       ELSE // illegal OPM              
           #FML_REF.OutData.FHPP[4] := 0;
           #Converted_BYTE5_8 := 0;
   END_CASE;

   (* Set Output DATA OF DRIVE *)
   #FML_REF.OutData.FHPP[5] := #BByte[1];
   #FML_REF.OutData.FHPP[6] := #BByte[2];
   #FML_REF.OutData.FHPP[7] := #BByte[3];
   #FML_REF.OutData.FHPP[8] := #BByte[4];
END_FUNCTION_BLOCK

FUNCTION_BLOCK "FB205_FHPP_SETIO_PART"   // FB205, SCL
TITLE = FHPPP SETIO_PART
{ S7_Optimized_Access := 'FALSE' }
AUTHOR : FESTO
FAMILY : E-DRIVE
VERSION : 5.1
// Set data from FHPP device using system function SETIO_PART
   VAR_INPUT
      ID : Word;
      Offset : Int;   // offset from start address where FHPP data start
   END_VAR
   VAR_OUTPUT
      Error : Bool;   // error while reading
      Status : "DT_FML_STATUS";
   END_VAR
   VAR_IN_OUT
      FML_REF : "DT_FML_REF";
   END_VAR
   VAR
      SET_PART : SETIO_PART;
   END_VAR
   VAR_TEMP
      i : Int;
      iByteCount : DInt;
      tmpFHPPplusSize : DInt;
      tmpFHPPplusElementSize : Array[1..9] of DInt;
      FHPPplus24 : Array[1..24] of Byte;
      WORD_BYTE : Word;
      WBYTE AT WORD_BYTE : Array[1..2] of Byte;
      DWORD_BYTE : DInt;
      DBYTE AT DWORD_BYTE : Array[1..4] of Byte;
      tmpStatus : "DT_FML_STATUS";
      tmp_FML_REF : "DT_FML_REF";
   END_VAR
BEGIN
   (*############################################################
       FESTO AG  Co., Esslingen
       Copyright (c) 2015. All rights reserved.    

       NAME OF FUNCTION BLOCK:         FHPP_SETIO_PART
       VERSION NUMBER:                 V5.1
       COMPOSER:                       bejk

   ############################################################*)

   // function block (FB) is busy
   #tmpStatus.Err := FALSE;
   #tmpStatus.Cat := 1;
   #tmpStatus.ID := 16#0000_0002; // FB busy 

   // ### FHPP Standard ###########################################
   #SET_PART(ID := #ID,
             OFFSET := #Offset,
             LEN := 8,
             ERROR => #tmpStatus.Err,
             OUTPUTS := #FML_REF.OutData.FHPP);

   // Error while writing
   IF #tmpStatus.Err THEN
       #tmpStatus.Cat := 4; // SIEMENS
       #tmpStatus.ID := DWORD_TO_DINT(#SET_PART.STATUS);
   END_IF;



   // ### EXIT ROUTINE ############################################################
   IF NOT #tmpStatus.Err THEN
       ENO := TRUE;      // Set ENO-Bit to true
       #Status := #tmpStatus;
       #Error := #tmpStatus.Err;
   ELSE
       ENO := FALSE;     // Set ENO-Bit to false
       #Status := #tmpStatus;
       #Error := #tmpStatus.Err;
   END_IF;
END_FUNCTION_BLOCK

FUNCTION "FC201_FPC_MAPPING" : Bool   // FC201, SCL
TITLE = FPC Mapping
{ S7_Optimized_Access := 'FALSE' }
AUTHOR : FESTO
FAMILY : E-DRIVE
VERSION : 5.1
// data mapping for parameter channel
   VAR_INPUT
      Mode : Bool;   // FALSE = MAP INPUTS/ TRUE = MAP OUTPUTS
   END_VAR
   VAR_IN_OUT
      FML_REF : "DT_FML_REF";
   END_VAR
   VAR_TEMP
      _Word : Word;
      BByte2 AT _Word : Array[1..2] of Byte;
      _DINT : DInt;
      BByte4 AT _DINT : Array[1..4] of Byte;
      Req_Identifier : Int;
      Resp_Identifier : Int;
   END_VAR
   VAR CONSTANT
      Const_1 : Byte := 1;
      Const_4 : Byte := 4;
   END_VAR
BEGIN
   (*############################################################
      FESTO AG  Co., Esslingen
      Copyright (c) 2015. All rights reserved.    

      NAME OF FUNCTION BLOCK:         FPC_MAPPING
      VERSION NUMBER:                 V5.1
      COMPOSER:                       bejk

   -----------------------------------------------------
      Date        Name                Activity                                                                              
      06.08.2015  Benjamin Kilgus     created (V1.0)
      07.07.2017  Benjamin Klein      version changed (V5.1)
      17.11.2017  Benjamin Klein      resp_identifier enhanced for SFC and MTR
   ############################################################*)

   (* MAP INPUTS *)
   IF NOT #Mode THEN

       // Byte1 FPCS            
       #FML_REF.FPCS_Modus := SHR(IN := (#FML_REF.InData.FPC[1] AND 2#11110000), N := 4);

       // decoding of EFPC modus
       CASE BYTE_TO_INT(#FML_REF.FPCS_Modus) OF
           0: (* old style *)
               (* 
               -------------- Byte 1 --------------- Byte 2 ---------------------- Byte 3/4 ------------------- Byte 5..8 ----
               |  8  7  6  5  4  |  3  2  1  0  |              | 15 14 13 12 |  11  | 10 9 8 7 6 5 4 3 2 1 0 |               |
               |    FPCS Modus   |     res      |   Subindex   |      AK     |  SPM |        PNU             |     Value     |
               ---------------------------------------------------------------------------------------------------------------     
               AK:  Response Identifier (Antwortkennung)
               SPM: NOT used
               PNU: Parameternummer / Parameter-Number 
               *)
               // Byte1
               // zero in this CASE
               // Byte2  
               #FML_REF.ActSubindex := #FML_REF.InData.FPC[2];

               // Byte3/4
               #BByte2[1] := #FML_REF.InData.FPC[3];
               #BByte2[2] := #FML_REF.InData.FPC[4];
               #Resp_Identifier := WORD_TO_INT(SHR(IN := (#_Word AND 2#1111000000000000), N := 12));
               #FML_REF.ActPNU := #_Word AND 2#0000011111111111;

               // Byte 5..8 parameter value
               #BByte4[1] := #FML_REF.InData.FPC[5];
               #BByte4[2] := #FML_REF.InData.FPC[6];
               #BByte4[3] := #FML_REF.InData.FPC[7];
               #BByte4[4] := #FML_REF.InData.FPC[8];
               #FML_REF.ParamValueRD := #_DINT;

           1, 2, 3:(* modus: 1 = PNU extended; 2 = KO; 3 = CAN Objects *)
               (* 
               -------------- Byte 1 --------------- Byte 2 ------------------- Byte 3/4----------------- Byte 5..8 ----
               |   7  6  5  4  |  3  2  1  0  |              | 15 14 13 12 11 10 9 8 7 6 5 4 3 2 1 0 |               |
               |  FPCS Modus   |     AK       |   Subindex   |   PNU extended or KO or CAN Object    |     Value     |
               -------------------------------------------------------------------------------------------------------       
               AK:  Response Identifier (Antwortkennung)
               *)

               // Byte 1 FPCS
               #Resp_Identifier := WORD_TO_INT(#FML_REF.InData.FPC[1] AND 2#00001111);

               // Byte 2 Subindex
               #FML_REF.ActSubindex := #FML_REF.InData.FPC[2];

               // Byte 3+4 **PKE/ PNU/ KO/ CAN**
               #BByte2[1] := #FML_REF.InData.FPC[3];
               #BByte2[2] := #FML_REF.InData.FPC[4];
               #FML_REF.ActPNU := #_Word;

               // Byte 5..8 parameter value
               #BByte4[1] := #FML_REF.InData.FPC[5];
               #BByte4[2] := #FML_REF.InData.FPC[6];
               #BByte4[3] := #FML_REF.InData.FPC[7];
               #BByte4[4] := #FML_REF.InData.FPC[8];
               #FML_REF.ParamValueRD := #_DINT;

           4, 5:(* FPCS_Modus 4=Parameter File; 5=Firmware File *)
               (*
               ------ BYTE 1 ------------|-- BYTE 2 -|--BYTE 3..8 ---|
               | 7  6  5  4 | 3  2  1  0 |           |               |
               | FPCS Modus |   res      | Packet-ID |  6 BYTE Data  |
               -------------------------------------------------------        
                 Packet-ID: -------------- BYTE 2 ----------
                            | 7    6    5  | 4  3  2  1  0 |
                            | Control Bits |   Sequence-Nr |
                            -------------------------------- 
               *)
               // Byte 1 FPCS
               #Resp_Identifier := WORD_TO_INT(#FML_REF.InData.FPC[1] AND 2#00001111);
               #FML_REF.RespID := #Resp_Identifier;

               //---- Byte 2 Packet-ID ----    
               #FML_REF.FPCS_Packet.BitSequenceNr := WORD_TO_INT(#FML_REF.InData.FPC[2] AND 2#00011111);
               #FML_REF.FPCS_Packet.Control := WORD_TO_INT(SHR(IN := (#FML_REF.InData.FPC[2] AND 2#11100000), N := 5));
               //---- Byte 3..8 Data ----
               #FML_REF.FPCS_Packet.Data[1] := #FML_REF.InData.FPC[3];
               #FML_REF.FPCS_Packet.Data[2] := #FML_REF.InData.FPC[4];
               #FML_REF.FPCS_Packet.Data[3] := #FML_REF.InData.FPC[5];
               #FML_REF.FPCS_Packet.Data[4] := #FML_REF.InData.FPC[6];
               #FML_REF.FPCS_Packet.Data[5] := #FML_REF.InData.FPC[7];
               #FML_REF.FPCS_Packet.Data[6] := #FML_REF.InData.FPC[8];


           ELSE (* not implemented *)
               #FC201_FPC_MAPPING := FALSE; (* Execution was not correct *)
               RETURN;
       END_CASE;

       CASE #Resp_Identifier OF
           0, 3:(* No Transmission or Active*)
               #FML_REF.Done := FALSE;
               #FML_REF.Err := FALSE;
               #FML_REF.ActPNU := 0;
               #FML_REF.ActSubindex := 0;
               #FML_REF.ParamValueRD := 0;
               #FML_REF.DatatypeRD := 0;


           1, 4:(* Word Parameter transmittead*)
               #FML_REF.Done := TRUE;
               #FML_REF.Err := FALSE;
               #FML_REF.ParamValueRD := #_DINT;
               #FML_REF.DatatypeRD := 2;

           2, 5: (*DWord Parameter transmitted*)
               #FML_REF.Done := true;
               #FML_REF.Err := FALSE;
               #FML_REF.ParamValueRD := #_DINT;
               #FML_REF.DatatypeRD := 4;

           7:(* Transmission Failed*)
               #FML_REF.Done := TRUE;
               #FML_REF.Err := TRUE;
               #FML_REF.DatatypeRD := 0;
               #FML_REF.ParamValueRD := 0;
               #FML_REF.ActPNU := 0;


           11, 12: (*BYTE Parameter transmitted*)
               #FML_REF.Done := TRUE;
               #FML_REF.Err := False;
               #FML_REF.DatatypeRD := 1;
               #FML_REF.ParamValueRD := #_DINT;

           ELSE (* not specified*)
               #FML_REF.Done := false;
               #FML_REF.Err := TRUE;
               #FML_REF.ParamValueRD := 0;
       END_CASE;

       #FC201_FPC_MAPPING := TRUE; (* Execution was correct *)
       RETURN;

   (* MAP OUTPUTS *)
   ELSE

       IF #FML_REF.DeviceTypeNo = 70 OR #FML_REF.DeviceTypeNo = 80 THEN
           IF #FML_REF.ReqID = 8 THEN // write
               IF BYTE_TO_INT(#FML_REF.Subindex) > 0 THEN
                   CASE BYTE_TO_INT(#FML_REF.DatatypeWR) OF
                       1:
                           #FML_REF.ReqID := 12;     //Array-Byte
                       2:
                           #FML_REF.ReqID := 7;      //Array-Wort
                       4:
                           #FML_REF.ReqID := 8;      //Array-Doppelwort
                       ELSE
                           #FC201_FPC_MAPPING := FALSE; (* wrong data type*)
                           RETURN;
                   END_CASE;
               END_IF;
               (*WRITE SINGLE PARAMETER*)
               IF #FML_REF.Subindex = 0 THEN
                   CASE BYTE_TO_INT(#FML_REF.DatatypeWR) OF
                       1:
                           #FML_REF.ReqID := 11;       // Single-Byte
                       2:
                           #FML_REF.ReqID := 2;        // Single-Wort
                       4:
                           #FML_REF.ReqID := 3;        // Single-Doppelwort
                       ELSE
                           #FC201_FPC_MAPPING := FALSE; (* wrong data type*)
                           RETURN;
                   END_CASE;
               END_IF;

           ELSIF #FML_REF.ReqID = 6 THEN
               (* READ ARRAY PARAMETER *)
               IF BYTE_TO_INT(#FML_REF.Subindex) > 0 THEN
                   #FML_REF.ReqID := 6;
               END_IF;
               (* READ SINGLE PARAMETER *)
               IF #FML_REF.Subindex = 0 THEN
                   #FML_REF.ReqID := 1;
               END_IF;
           ELSE
               ;// not specified
           END_IF;
       END_IF;
       (* create request identifier *)
       #Req_Identifier := #FML_REF.ReqID;

       CASE BYTE_TO_INT(#FML_REF.FPCC_Modus) OF
           0: (* old style *)
               (* 
               -------------- Byte 1 --------------- Byte 2 ---------------------- Byte 3 --------------------- Byte 5..8 ----
               |  8  7  6  5  4  |  3  2  1  0  |              | 15 14 13 12 |  11  | 10 9 8 7 6 5 4 3 2 1 0 |               |
               |    FPCS Modus   |     res      |   Subindex   |      AK     |  SPM |        PNU             |     Value     |
               ---------------------------------------------------------------------------------------------------------------     
               AK:  Request Identifier (Auftragskennung)
               SPM: NOT used
               PNU: Parameternummer / Parameter-Number 
               *)
               (* Byte 1 *)
               #FML_REF.OutData.FPC[1] := SHL(IN := #FML_REF.FPCC_Modus, N := 4);
               (* Byte 2 Subindex *)
               #FML_REF.OutData.FPC[2] := #FML_REF.Subindex;
               (* Byte 3+4 *)
               #_Word := SHL(IN := INT_TO_WORD(#Req_Identifier), N := 12) OR (#FML_REF.PNU AND 16#07_FF);

               (* Byte 5..8 *)
               #_DINT := #FML_REF.ParamValueWR;
               #FML_REF.OutData.FPC[3] := #BByte2[1]; //Convert PKE to Byte
               #FML_REF.OutData.FPC[4] := #BByte2[2];

               (* Set Output DATA OF DRIVE *)
               #FML_REF.OutData.FPC[5] := #BByte4[1]; //Convert PWE to Byte
               #FML_REF.OutData.FPC[6] := #BByte4[2];
               #FML_REF.OutData.FPC[7] := #BByte4[3];
               #FML_REF.OutData.FPC[8] := #BByte4[4];

           1, 2, 3:(* modus: 1 = PNU extended; 2 = KO; 3 = CAN Objects *)
               (* 
               -------------- Byte 1 --------------- Byte 2 ------------------- Byte 3 ------------------ Byte 5..8 ----
               |  8  7  6  5  4  |  3  2  1  0  |              | 15 14 13 12 11 10 9 8 7 6 5 4 3 2 1 0 |               |
               |    FPCS Modus   |     AK       |   Subindex   |   PNU extended or KO or CAN Object    |     Value     |
               ---------------------------------------------------------------------------------------------------------       
               AK:  Request Identifier (Auftragskennung)
               *)
               (* Byte 1 *)
               #FML_REF.OutData.FPC[1] := WORD_TO_BYTE(SHL(IN := #FML_REF.FPCC_Modus, N := 4) OR INT_TO_WORD(#Req_Identifier));
               (* Byte 2 Subindex *)
               #FML_REF.OutData.FPC[2] := #FML_REF.Subindex;
               (* Byte 3+4 *)
               #_Word := #FML_REF.PNU;
               (* Byte 5..8 *)
               #_DINT := #FML_REF.ParamValueWR;
               #FML_REF.OutData.FPC[3] := #BByte2[1]; //Convert PKE to Byte
               #FML_REF.OutData.FPC[4] := #BByte2[2];

               (* Set Output DATA OF DRIVE *)
               #FML_REF.OutData.FPC[5] := #BByte4[1]; //Convert PWE to Byte
               #FML_REF.OutData.FPC[6] := #BByte4[2];
               #FML_REF.OutData.FPC[7] := #BByte4[3];
               #FML_REF.OutData.FPC[8] := #BByte4[4];

           4, 5:(* FPCC_Modus 4=parameter file; 5=firmware file     
           |---------- byte 1 --------|-- byte 2 --|-- byte 3..8 ---|
           | 7  6  5  4  | 3  2  1  0 |            |                |
           |   FPCC modus |   res      | packet-ID  |  6 byte data  |
           ---------------------------------------------------------       
           Packet-ID:  | 7    6    5  | 4  3  2  1  0  |
                       | control bits |  sequence-nr   |
                       --------------------------------- *)
                       //---- byte 1 ----
                       #FML_REF.OutData.FPC[1] := WORD_TO_BYTE(SHL(IN := #FML_REF.FPCC_Modus, N := 4) OR INT_TO_WORD(#Req_Identifier));
                       //----byte 2 packet-ID ---- 
                       #FML_REF.OutData.FPC[2] := (SHL(IN := INT_TO_BYTE(#FML_REF.FPCC_Packet.Control), N := 5) OR (INT_TO_BYTE(#FML_REF.FPCC_Packet.BitSequenceNr) AND 16#1F));
                       //---- byte 3..8 data ----
                       #FML_REF.OutData.FPC[3] := #FML_REF.FPCC_Packet.Data[1];         // byte swapping for modbus data 
                       #FML_REF.OutData.FPC[4] := #FML_REF.FPCC_Packet.Data[2];
                       #FML_REF.OutData.FPC[5] := #FML_REF.FPCC_Packet.Data[3];
                       #FML_REF.OutData.FPC[6] := #FML_REF.FPCC_Packet.Data[4];
                       #FML_REF.OutData.FPC[7] := #FML_REF.FPCC_Packet.Data[5];
                       #FML_REF.OutData.FPC[8] := #FML_REF.FPCC_Packet.Data[6];

                   ELSE (* not implemented *)
                       #FC201_FPC_MAPPING := FALSE; (* Execution was not correct *)
                       RETURN;
               END_CASE;

               #FC201_FPC_MAPPING := TRUE; (* Execution was correct *)
           END_IF;
END_FUNCTION

FUNCTION "FC202_FHPPPLUS_MAPPING" : DInt   // FC202, SCL
TITLE = FHPPPLUS_MAPPING
{ S7_Optimized_Access := 'FALSE' }
AUTHOR : FESTO
FAMILY : E-DRIVES
VERSION : 5.1
// data mapping for FHPPplus data
   VAR_INPUT
      cfgFHPPplus : DInt;
   END_VAR
   VAR_OUTPUT
      FHPPplusElementSize : Array[1..9] of DInt;
      FHPPplusSize : DInt;
   END_VAR
   VAR_TEMP
      i : Int;
      n : Int;
      tmpTeiler : DInt;
      tmpCfgFHPPplus : DInt;
      tmpElementSize : DInt;
      tmpFHPPplusSize : DInt;
   END_VAR
   VAR CONSTANT
      constTeiler : DInt := 100_000_000;
   END_VAR
BEGIN
   (*############################################################
      FESTO AG  Co., Esslingen
      Copyright (c) 2015. All rights reserved.    

      NAME OF FUNCTION BLOCK:         FHPPPLUS_MAPPING
      VERSION NUMBER:                 V5.1
      COMPOSER:                       bejk

      LAST CHANGE:                    06.08.2015

      -----------------------------------------------------
      Date        Name                Activity                                                                              
      06.08.2015  Benjamin Kilgus     created (V1.0)
      29.08.2016  Benjamin Klein      version changed (V4.1)
      05.07.2017  Benjamin Klein      changed to optimized access (V5.1)

   ############################################################*)

   #tmpTeiler := #constTeiler;
   #tmpCfgFHPPplus := #cfgFHPPplus;
   #tmpFHPPplusSize := 0;
   #n := 1;

   // configuration 0 is not legal
   IF #cfgFHPPplus = 0 THEN
       #FC202_FHPPPLUS_MAPPING := DWORD_TO_DINT(16#8000_0001);
       RETURN;
   END_IF;

   FOR #i := 1 TO 9 DO
       #tmpElementSize := #tmpCfgFHPPplus / #tmpTeiler;
       IF #tmpElementSize = 1 OR #tmpElementSize = 2 OR #tmpElementSize = 4 THEN
           #FHPPplusElementSize[#n] := #tmpElementSize * 8; // Byte *8 = Bit
           #tmpFHPPplusSize := #tmpFHPPplusSize + #FHPPplusElementSize[#n];
           #tmpCfgFHPPplus := #tmpCfgFHPPplus - (#tmpElementSize * #tmpTeiler);
           #n := #n + 1;
       ELSIF #tmpElementSize = 0 AND #n = 1 THEN // digit empty
           #FHPPplusElementSize[10 - #i] := 0;
       ELSE
           #FC202_FHPPPLUS_MAPPING := DWORD_TO_DINT(16#8000_0001); // wrong configuration
           RETURN;
       END_IF;
       #tmpTeiler := #tmpTeiler / 10;
   END_FOR;

   IF #tmpFHPPplusSize = 64 OR #tmpFHPPplusSize = 128 OR #tmpFHPPplusSize = 192 THEN
       ;// o.k.

   ELSE // wrong size
       #FC202_FHPPPLUS_MAPPING := DWORD_TO_DINT(16#8000_0001); // function is called without legal FHPP+ configuration
       RETURN;
   END_IF;

   #FHPPplusSize := #tmpFHPPplusSize;
   #FC202_FHPPPLUS_MAPPING := 0; // o.k.
END_FUNCTION

// folder: 03_Pgv/01_Function

FUNCTION_BLOCK "FB301_PgvDados"   // FB4, SCL
{ S7_Optimized_Access := 'FALSE' }
VERSION : 0.1
// Este bloco realiza a troca de dados do AGV com o PGV
   VAR
      Pgv_Escrita : Struct   // Saida de dados de escrita
         LADDR : Word := W#16#1;   // Endereço do PGV
         RECORD : String := '';   // Endereço de escrita da informação no PGV
         RET_VAL : Int;   // Codigo de erros
      END_STRUCT;
      Pgv_Leitura : Struct   // Saida de dados de leitura
         LADDR : Word := W#16#1;   // Endereço do PGV
         RECORD : String;   // Endereço de escrita da informação no PGV
         RET_VAL : Int;   // Codigo de erros
      END_STRUCT;
   END_VAR
BEGIN
   (*
       Este bloco realiza a troca de dados do AGV com o PGV
   *)

   REGION EscreveDadosPGV
       #Pgv_Escrita.RET_VAL := DPWR_DAT(LADDR := #Pgv_Escrita.LADDR, RECORD :=  P#DB1.DBX285.0 byte 1);
   END_REGION

   REGION LeituraDadosPGV
       //#Pgv_Leitura.RET_VAL := DPRD_DAT(LADDR := #Pgv_Leitura.LADDR, RECORD => P#DB1.DBX8.0 byte 14);
       "DB1_DatabaseAgv".PGV.Module2.Status.ERR := "ERR";
       "DB1_DatabaseAgv".PGV.Module2.Status.NP := "NP";
       "DB1_DatabaseAgv".PGV.Module2.Status.WRN := "WRN";
       "DB1_DatabaseAgv".PGV.Module2.Status.CC := "CC";
       "DB1_DatabaseAgv".PGV.Module2.Status.Reservado := "Reservado";
       "DB1_DatabaseAgv".PGV.Module2.Status.FR := "FR";
       "DB1_DatabaseAgv".PGV.Module2.Status.FL := "FL";
       "DB1_DatabaseAgv".PGV.Module2.Status.NL := "NL";
       "DB1_DatabaseAgv".PGV.Module2.Status.RP := "RP";
       "DB1_DatabaseAgv".PGV.Module2.Status.LC := "LC";
       "DB1_DatabaseAgv".PGV.Module2.Status.LC_1 := "LC_1";
       "DB1_DatabaseAgv".PGV.Module2.Status.TA := "TA";
       "DB1_DatabaseAgv".PGV.Module2.Status.Reservado_1 := "Reservado_1";
       "DB1_DatabaseAgv".PGV.Module2.Status.Reservado_2 := "Reservado_2";
       "DB1_DatabaseAgv".PGV.Module2.Status.Reservado_3 := "Reservado_3";
       "DB1_DatabaseAgv".PGV.Module2.Status.Reservado_4 := "Reservado_4";
       "DB1_DatabaseAgv".PGV.Module2.PositionY := "PositionY";
       "DB1_DatabaseAgv".PGV.Module2.Angle := "Angle";
       "DB1_DatabaseAgv".PGV.Module2.PositionX := "PositionX";
       "DB1_DatabaseAgv".PGV.Module2.PositionZ := "PositionZ";
       "DB1_DatabaseAgv".PGV.Module5.Status := "Status";
       "DB1_DatabaseAgv".PGV.Module5.BitmaskWarning := "Status";
       "DB1_DatabaseAgv".PGV.Module5.ErroNumber := "Erro";
   END_REGION
END_FUNCTION_BLOCK

FUNCTION_BLOCK "FB300_LogicaPgv"   // FB300, SCL
TITLE = FB300_LogicaPgv
{ S7_Optimized_Access := 'FALSE' }
AUTHOR : ssbjvq
FAMILY : AGV_KD
VERSION : 0.1
// Este bloco controla a logica de direção do AGV, lendo os dados do PGV e os processando por meio de um controle proporcional.
   VAR_INPUT
      In_PosicaoY : DWord;   // Valor de posicionamento no eixo y
      In_Angulo : Word;   // Valor de angulo
      In_ForaRota : Bool;   // Sinal de fora da rota
      In_Emergencia : Bool;   // Sinal de emergencia AGV
      In_ManAuto : Int;   // Sinal de Modo de operação Man/Aut
      In_Start : Bool;   // Sinal da memoria Start
      In_RotaEscolhida : Byte;   // Sinal de rota/Processo escolhido, vindo da IHM
   END_VAR
   VAR_OUTPUT
      Out_Angulo : Int;   // Valor de Angulo com filtro
      Out_Direita : Bool;   // Acionamento Direita
      Out_Esquerda : Bool;   // Acionamento Esquerda
      Out_NaRota : Bool;   // Sinal de verificação de AGV na rota
      Out_EmCurva : Bool;   // Sinal de AGV em curva brusca
      Out_EmCurvaIntermedio : Bool;   // Sinal de AGV em curva intermediaria/leve
      Out_ProcessoEscolhido : Int;   // Sinal de processo escolhido
   END_VAR
   VAR
      S_ResolucaoMaxima : Int := 32767;   // Memoria de valor de resolução maxima
      S_CalculoProporcional : Int;   // Memoria do valor do calculo proporcional
      S_Angulo : Int;   // Memoria do Angulo convertido
      S_PosicaoY : Int;   // Memoria da posição Y
      S_Direita : Bool;   // Memoria acionamento direta
      S_Esquerda : Bool;   // Memoria acionamento esquerda
      S_NaRota : Bool;   // Memoria de AGV na rota
      S_EmCurva : Bool;   // Memoria AGV em curva
      S_EmCurvaIntermedio : Bool;   // Memoria AGV em curva
   END_VAR
BEGIN
   (*
       Este bloco controla a logica de direção do AGV, lendo os dados do PGV e os processando por meio de um controle proporcional. 
   *)

   REGION ConversãoDeValores
       //Realização de conversão e formatação de valores
       #S_Angulo := WORD_TO_INT(#In_Angulo);
       #S_PosicaoY := DWORD_TO_INT(#In_PosicaoY);

   END_REGION

   REGION Temporizadores
       //Temporizador que identifica que o AGV está fora da rota
       "TOF_ParaAgv".TOF(IN := (#S_PosicaoY = 999),
                         PT := T#1s);
   END_REGION

   //Contém a logica de controle do AGV
   REGION LogicaDeControle
       //Verifica se está fora da rota
       IF #In_ForaRota AND NOT (#S_PosicaoY = 999) THEN
           #S_NaRota := 1;
       ELSE
           #S_NaRota := 0;
       END_IF;
       //Verifica se o emergencia está acionado
       IF #In_Emergencia THEN
           //Verifica se está fora da rota e se esta em modo automatico
           IF NOT (#S_PosicaoY = 999) AND (#In_ManAuto = 2) THEN
               #S_CalculoProporcional := #S_PosicaoY;
               //Entre 50 e -50 o AGV não atual a correção
               IF #S_CalculoProporcional > 55 THEN
                   //Entre 75 e 85 identifica uma curva/variação intermediaria
                   IF #S_CalculoProporcional > 70 AND #S_CalculoProporcional <= 85 THEN
                       #S_EmCurvaIntermedio := 1;
                       #S_EmCurva := 0;
                   //Entre 85 identifica uma curva/variação brusca
                   ELSIF #S_CalculoProporcional > 85 THEN
                       #S_EmCurvaIntermedio := 0;
                       #S_EmCurva := 1;
                   ELSE
                       #S_EmCurva := 0;
                       #S_EmCurvaIntermedio := 0;
                   END_IF;
                   #S_Direita := 1;
                   #S_Esquerda := 0;
                   //Entre 50 e -50 o AGV não atual a correção
               ELSIF #S_CalculoProporcional < -55 THEN
                   //Entre -75 e -85 identifica uma curva/variação intermediaria
                   IF #S_CalculoProporcional > -85 AND #S_CalculoProporcional < -70 THEN
                       #S_EmCurvaIntermedio := 1;
                       #S_EmCurva := 0;
                   //Entre -85 identifica uma curva/variação brusca  
                   ELSIF #S_CalculoProporcional < -85 THEN
                       #S_EmCurvaIntermedio := 0;
                       #S_EmCurva := 1;
                   ELSE
                       #S_EmCurvaIntermedio := 0;
                       #S_EmCurva := 0;
                   END_IF;
                   #S_Direita := 0;
                   #S_Esquerda := 1;
               ELSE
                   #S_Direita := 0;
                   #S_Esquerda := 0;
               END_IF;
           ELSE
               #S_EmCurva := 0;
               #S_Direita := 0;
               #S_Esquerda := 0;
               #S_CalculoProporcional := 999;
           END_IF;
       ELSE
           #S_EmCurva := 0;
           #S_Direita := 0;
           #S_Esquerda := 0;
           #S_CalculoProporcional := 999;
       END_IF;
   END_REGION



   REGION Outputs
       // Coloca valores das memorias nas saidas
       #Out_EmCurva := #S_EmCurva;
       #Out_NaRota := #S_NaRota;
       #Out_Direita := #S_Direita;
       #Out_Esquerda := #S_Esquerda;
       #Out_EmCurvaIntermedio := #S_EmCurvaIntermedio;
       #Out_ProcessoEscolhido := BYTE_TO_INT(#In_RotaEscolhida);

   END_REGION
END_FUNCTION_BLOCK

// folder: 04_Rfid/01_Function

FUNCTION_BLOCK "FB400_LogicaRfid"   // FB400, SCL
TITLE = FB400_LogicaRfid
{ S7_Optimized_Access := 'FALSE' }
AUTHOR : ssbjvq
FAMILY : AGV_KD
VERSION : 1.0
// Este bloco controla do a logica de valores de parada, velocidade e posto. estes valores são lidos de um cartão RFID pela antena RFID no AGV.
   VAR_INPUT
      In_ManAuto : Int;   // Sinal de modo aut/man
      In_LeituraEscrita : Int;   // Sinal de modo do RFID, vindo da IHM - 1 = Leitura / 2 = Escrita
      In_Comando : Int;   // Sinal de comando vindo da DB do AGV
      In_OldComando : Int;   // Sinal de velho comando vindo da DB do AGV
      In_Velocidade : Int;   // Sinal de Vel vindo da DB do AGV
      In_Linha : Int;   // Sinal de Linha vindo da DB do AGV
      In_Posto : Int;   // Sinal de Posto vindo da DB do AGV
      In_TagPresente : Bool;   // Sinal de tag presente
      In_HmiProcesso : Int;   // Valor de qual linha foi escolhida para o AGV rodar e obedecer as Tags // 1 - ECU / 10 - SKD
      In_GravaPosto : Int;   // Valor de gravação de tag
      In_GravaComando : Int;   // Valor de gravação de tag
      In_GravaVel : Int;   // Valor de gravação de tag
      In_GravaProcesso : Int;   // Valor de gravação de tag
   END_VAR
   VAR_OUTPUT
      Out_PararAgv : Bool;   // Sinal que faz a parada do AGV
      Out_Comando : Int;   // Sinal que exporta o comando do AGV
      Out_Velocidade : Int;   // Sinal que exporta a velocidade do AGV
      Out_Linha : Int;   // Sinal que exporta qual linha a tag representa
      Out_Posto : Int;   // Sinal que exporta posto que o AGV está
      Out_LeituraEscrita : Int;   // Sinal que exporta o modo do RFID
      Out_GravaPosto : Int;   // Sinal de gravação de posto na tag
      Out_GravaComando : Int;   // Sinal de gravação de Comando na tag
      Out_GravaVel : Int;   // Sinal de gravação de Vel na tag
      Out_GravaProcesso : Int;   // Sinal de gravação de Linha na tag
   END_VAR
   VAR
      TOF_Rfid : TOF;   // Temporizador que faz o reset do comando de parada, após o AGV parar na tag.
      S_ParaAgv : Bool;   // Memoria que faz o AGV para na tag
      Balluff_Rfid_Instance : "FB401_Balluff_Rfid";   // Este bloco é criado e parametrizado para fazer a leitura dos dados da antena RFID
      TimerResetError : TON;   // Este temporizador verifica se o RFID tem algum erro ou não esta pronto para atuar na leitura e soluciona o problema de falha ou mal funcionamento
      TON_RFID : TON;   // Temporizador de filtro, que so realiza o acionamento quando a tag ta presente por 100ms.
   END_VAR
BEGIN
   (*
     Este bloco controla do a logica de valores de parada, 
     velocidade e posto. estes valores são lidos de um cartão 
     RFID pela antena RFID no AGV. 
   *)

   //Temporizadores utilizados na logica
   REGION Temporizadores
       //Temporizador de filtro, que so realiza o acionamento quando a tag ta presente por 100ms.
       #TON_RFID(IN := #In_TagPresente,
                 PT := T#100ms);
       //Temporizador que faz o reset do comando de parada, após o AGV parar na tag.
       #TOF_Rfid(IN := #In_TagPresente AND (#In_Comando = 1),
                 PT := T#2s);
   END_REGION

   //Logica não utilizada
   REGION LogicaComentada
       //Era utiliza para fazer com que o AGV parasse em todas as tags, independente do comando.
       (* IF #TOF_Rfid.Q THEN
               #S_ParaAgv := 1;
          ELSE
               #S_ParaAgv := 0;
          END_IF; *)
   END_REGION

   //Contém a logica principal do bloco 
   REGION Logica
       //Logica em Modo Leitura
       IF #In_ManAuto = 2 AND #In_LeituraEscrita = 1 THEN
           //Verifica a tag presente e o temporizador
           IF (#In_TagPresente OR #TOF_Rfid.Q) THEN
               //Verifica o comando
               IF #In_Comando = 1 AND (#In_Linha = #In_HmiProcesso) THEN
                   IF #TOF_Rfid.ET >= T#1.8s THEN
                       "DB420_LeituraRfid".RfidLeitura[2] := 0;
                   END_IF;
                   #S_ParaAgv := 1;
               ELSE
                   #S_ParaAgv := 0;
               END_IF;
               //Coloca os valores lidos e processado na saida do bloco.
               #Out_Comando := #In_Comando;
               #Out_Velocidade := #In_Velocidade;
               #Out_Linha := #In_Linha;
               #Out_Posto := #In_Posto;

           ELSE
               #S_ParaAgv := 0;
           END_IF;
       //Logica para quando o Modo Gravação de tag está ativada
       ELSIF #In_LeituraEscrita = 2 THEN
           #Out_GravaPosto := #In_GravaPosto;
           #Out_GravaComando := #In_GravaComando;
           #Out_GravaVel := #In_GravaVel;
           #Out_GravaProcesso := #In_GravaProcesso;
       ELSE
           #Out_Comando := #In_Comando;
           #Out_Velocidade := #In_Velocidade;
           #Out_Linha := #In_Linha;
           #Out_Posto := #In_Posto;
           #Out_PararAgv := 0;
       END_IF;
       #Out_PararAgv := #S_ParaAgv;
   END_REGION









   REGION BlocoDeControleDoRfid
       (*
           Este bloco é criado e parametrizado para fazer a leitura dos dados da antena RFID
       *)
       #Balluff_Rfid_Instance(Init := "DB1_DatabaseAgv".RFID.Inputs.Init,
                              Start := "DB1_DatabaseAgv".RFID.TagPresente,
                              Reset := "DB1_DatabaseAgv".RFID.Inputs.Reset,
                              HeadOff := "DB1_DatabaseAgv".RFID.Inputs.HeadOff,
                              Dynamic := "DB1_DatabaseAgv".RFID.Inputs.Dynamic,
                              "HW_IO" := "DB1_DatabaseAgv".RFID.Inputs."HW_IO",
                              Command := "DB1_DatabaseAgv".RFID.Inputs.Command,
                              DB_Send := "DB1_DatabaseAgv".RFID.Inputs.DB_Send,
                              Offset_DBSend := "DB1_DatabaseAgv".RFID.Inputs.Offset_DBSend,
                              DB_Receive := "DB1_DatabaseAgv".RFID.Inputs.DB_Receive,
                              Offset_DBReceive := "DB1_DatabaseAgv".RFID.Inputs.Offset_DBReceive,
                              StartAddress := "DB1_DatabaseAgv".RFID.Inputs.StartAddress,
                              NumberOfByte := "DB1_DatabaseAgv".RFID.Inputs.NumberOfByte,
                              Watchdog := "DB1_DatabaseAgv".RFID.Inputs.Watchdog,
                              WD_Timer := #Balluff_Rfid_Instance.WD_Timer,
                              Ready => "DB1_DatabaseAgv".RFID.Ready,
                              Error => "DB1_DatabaseAgv".RFID.Error,
                              ErrorCode => "DB1_DatabaseAgv".RFID.CodigoErro,
                              DataCarrierPresent => "DB1_DatabaseAgv".RFID.TagPresente);

       "DB1_DatabaseAgv".RFID.Inputs.Init := "DB1_DatabaseAgv".RFID.Inputs.Init;


       //Este temporizador verifica se o RFID tem algum erro ou não esta pronto para atuar na leitura e soluciona o problema de falha ou mal funcionamento
       #TimerResetError(IN := ("DB1_DatabaseAgv".RFID.Error OR NOT "DB1_DatabaseAgv".RFID.Ready OR "DB500_SinaisIhm".ResetFalha_Rfid) AND #In_LeituraEscrita = 1,
                        PT := T#100ms,
                        Q => "DB1_DatabaseAgv".RFID.Inputs.Reset);
   END_REGION
END_FUNCTION_BLOCK

FUNCTION_BLOCK "FB401_Balluff_Rfid"   // FB401, STL
TITLE = Balluff RFID System BIS M IOLink with 32 Byte buffer (V1.1) / FB401_Balluff_Rfid
{ S7_Optimized_Access := 'FALSE' }
AUTHOR : Serrano
FAMILY : Ident
NAME : BISM_IOL
VERSION : 1.1
// Haftungsausschluss:
// *********************
// Der hier kostenlos verfügbare DEMO-Baustein ist ein allgemeingültiges 
// Anwendungsbeispiel. Dieser DEMO-Baustein soll bei der Programmierung und 
// Projektierung von SPS-Anwendungen unterstützen und Lösungsansätze aufzeigen. 
// Ein Anspruch auf Gewährleistung, Fehlerbeseitigung und Update besteht für den 
// Anwender nicht. Die BALLUFF GmbH schließt insbesondere jegliche Haftung für 
// Schäden, die durch den Einsatz dieses DEMO-Bausteins entstehen, ausdrücklich 
// aus! Diese Haftungsbeschränkung gilt nicht bei Verletzungen des Lebens, des 
// Körpers oder der Gesundheit, bei der Haftung nach dem Produkthaftungsgesetz und 
// bei vorsätzlichen Pflichtverletzungen. 
// Prüfen Sie vor dem Einsatz in Anlagen und Maschinen, ob der hier 
// bereitgestellte 
// DEMO Baustein für Ihre Anwendung nutzbar ist!
// Mit dem Einsatz des hier kostenlos vorgelegten S7-Beispiel erkennen Sie die 
// Gewährleistungs- und Haftungsbegrenzung an!
// 
// Disclaimer of Liability
// **********************
// The demo module made available here without cost is a generally accepted 
// example 
// application. This demo module shall support programming and conception of PLC 
// applications and shall provide possible methods of resolution.
// The user is not entitled to claim for warranty, fault clearance and updates. In 
// particular there is excluded any claims against Balluff GmbH for damages that 
// might result from the use of this demo module. Excluded from this limitation of 
// liability shall be (a) those damages that are based on injury to life, limb or 
// health, (b) a liability according to the Produkthaftungsgesetz (German Product 
// Liability Law) and (c) cases of wilful intent.
// Please check if the demo module is serviceable for your application before 
// adapting it in plants and machineries
// By using the S7 sample made available without cost you accept the limitation of 
// warranty and liability!
// 
// 
// BIS M 4XX-045-XXX-07-S4
// IO-Link Schnittstelle (V 1.1)
// Este bloco é criado e parametrizado para fazer a leitura dos dados da antena RFID
   VAR_INPUT
      Init : Bool;   // Internal reset and initailisation of FB
      Start : Bool;   // Start command
      Reset : Bool;   // Reset of BIS and FB
      HeadOff : Bool;   // Disable Antenna
      Dynamic : Bool;   // Dynamic read / write function
      HW_IO : Int;   // HW IO address of the module
      Command : Int;   // 1=Read;2=Write
      DB_Send : Int;   // Data block write data
      Offset_DBSend : Int;   // Offset of write data
      DB_Receive : Int;   // Data block for read data
      Offset_DBReceive : Int;   // Offset of data read
      StartAddress : Int;   // Start address from data carrier
      NumberOfByte : Int;   // data lenght to be written or read
      Watchdog : S5Time;   // Watchdog of function
      WD_Timer : Timer;   // Watchdog timer
   END_VAR
   VAR_OUTPUT
      Ready : Bool;   // Comamnd ready
      Error : Bool;   // Auftrag mit Fehler beendet
      ErrorCode : Int;   // Fehlernummer
      DataCarrierPresent : Bool;   // Data Carrier present
   END_VAR
   VAR
      EA_Laenge : Int;
      ZeigerByte : Int;   // Aktuelle Lese-/ Schreibadresse
      LaengeByte : Int;   // Anzahl Byte für Lese-/ Schreibzyklus
      ByteProSeite : Int;   // Anzahl maximaler Nutzbyte pro Seite
      Gesamtbyte : Int;   // Gesamtbyte die gelesen bzw. geschrieben werden
      LesenAktiv : Bool;   // Funktion Lesen ist aktiv
      SchreibenAktiv : Bool;   // Funktion Schreiben ist aktiv
      SchreibKonst : Bool;
      ResetAktiv : Bool;   // Funktion rücksetzen ist aktiv
      HeadOffAktiv : Bool;
      Toggle : Bool;   // Letzer Zustand des Toggle-Bit
      ErsterZyklus : Bool;   // Erster Schreib-/ Lesezyklus
      FP_Start : Bool;   // Flankenmerker Start
      IMP_Start : Bool;   // Impulsmerker Start
      FP_Reset : Bool;   // Flankenmerker Reset
      IMP_Reset : Bool;   // Impulsmerker Reset
      FP_CTPR : Bool;   // Flankenmerker Codetag-Present
      IMP_CTPR : Bool;   // Impulsmerker Codetag-Present
      CounterHF : Int;
      SeiteEingang : Array[0..31] of Byte;
      SeiteAusgang : Array[0..31] of Byte;
      Offset : Int;   // Instanz-DB Offset
      OffsetEin : Int;   // Offset Eingangsarray
      OffsetAus : Int;   // Offset Ausgangsarray
      IOAddress : Word;
   END_VAR
   VAR_TEMP
      InstanzDB : Int;   // Instanz-DB Nummer
      LOG_1 : Bool;   // Logisch 1
      Sp_start : Bool;   // Bei Fehler wird hier der Flankenmerker Start zwischengespeichert
      temp : Byte;   // Temporäre Variable
      schleife : Int;   // Schleifenzähler
      DB_Empf1 : Int;
      DB_Send1 : Int;
      ret : Int;
   END_VAR
BEGIN

REGION Network 1: SPS Anlauf
   // Initialisierung Instanz-Bereich
         AN    #LOG_1;
         S     #LOG_1;
         L     DINO;
         T     #InstanzDB;  // Nummer des Instanz-DB ermitteln
         OPN   DB[ #InstanzDB];
         TAR2;  // Bit-Offset des Instanz-DB
         SLD   8;
         SRD   8;
         L     8;
         /D;  // Offset Instanz-DB
         T     #Offset;
         L     42;
         +I;
         T     #OffsetEin;  // Offset des Eingangsarray
         L     #Offset;
         L     74;
         +I;
         T     #OffsetAus;  // Offset des Ausgangsarray

         L     #HW_IO;
         T     #IOAddress;

         L     32;
         T     #EA_Laenge;  // EA Länge Profibusmodul

         CALL  DPRD_DAT
         ( LADDR   := #IOAddress,
           RET_VAL := #ret,
           RECORD  := #SeiteEingang
         );

         L     #Offset;
         SLW   3;
         LAR1;

         AN    #Init;
         JC    M000;
         L     0;
         T     DBD[AR1, P#30.0];  //DBD30
         T     DBD[AR1, P#34.0];  //DBD34
         T     DBD[AR1, P#38.0];  //DBD38
         T     #ErrorCode;
         S     #Ready;
         R     #Error;
         R     #WD_Timer;
         BEU;
END_REGION

REGION Network 2: Kopfabschaltung
   M000: AN    #HeadOff;
         AN    #HeadOffAktiv;
         JC    M015;
         OPN   DB[ #InstanzDB];
         R     #LesenAktiv;
         R     #SchreibenAktiv;
         R     #SchreibKonst;
         R     #Toggle;
         R     #Error;
         L     0;
         T     #ZeigerByte;
         T     #Gesamtbyte;
         T     #ErrorCode;
         L     #OffsetEin;
         SLW   3;
         LAR1;
         A     DIX[AR1, P#0.6];  // HF-bit high
         O     #HeadOffAktiv;
         JC    M001;
         L     #OffsetAus;  // Offset Ausgangsarrey
         SLW   3;
         LAR1;
         L     0;
         T     DIB[AR1, P#0.0];  // Bitleiste rücksetzen
         A     #HeadOff;
         =     DIX[AR1, P#0.5];  // KA-bit setzen
         S     #HeadOffAktiv;
         R     #Ready;
         R     #DataCarrierPresent;
         JU    M002;
   M001: L     #OffsetEin;
         SLW   3;
         LAR1;
         A     #HeadOff;
         BEC;
         AN    DIX[AR1, P#0.6];  // HF-bit high
         JC    M003;
         L     #OffsetAus;
         SLW   3;
         LAR1;
         L     0;
         T     DIB[AR1, P#0.0];  // Bitleiste rücksetzen
   M002: L     DIB[AR1, P#0.0];  // 1. Bitleiste
         T     #temp;
         L     #OffsetAus;  // Adresse 2. Bitleiste
         L     #EA_Laenge;
         +I;
         L     1;
         -I;
         SLW   3;
         LAR1;
         L     #temp;
         T     DBB[AR1, P#0.0];
         JU    m100;
   M003: A     #LOG_1;
         R     #HeadOffAktiv;
         A     DIX[AR1, P#0.0];  // Datenträger vorhanden
         =     #DataCarrierPresent;
         BEU;
END_REGION

REGION Network 3: Eingangsdaten einlesen in Empfangs-DB
   // Bitleiste 1 einlesen in Instanz-DB
   M015: OPN   DB[ #InstanzDB];
         L     #OffsetEin;
         SLW   3;
         LAR1;  // Adresse Bitleiste 1 Pointerformat
         L     DBB[AR1, P#0.0];  // Bitleiste 1 einlesen
         T     #temp;

   // Bitleiste 2 einlesen in Instanz-DB
         L     #OffsetEin;
         L     #EA_Laenge;
         +I;
         L     1;
         -I;
         SLW   3;
         LAR1;  // Adresse Bitleiste 2 Pointerformat
         L     DBB[AR1, P#0.0];  // Bitleiste 2 einlesen
         L     #temp;
         <>I;
         BEC;  // Bitleisten unterschiedlich -> BEB
   // Fehlermeldungen abfragen
         AN    DIX[AR1, P#0.3];  //DIX42.3 Fehler vorhanden ?
         O     #Reset;  // oder Reset
         JC    wt1;
         L     #OffsetEin;
         L     1;
         +I;
         SLW   3;
         LAR1;
         L     DBB[AR1, P#0.0];  // Fehlernummer laden
         T     #ErrorCode;
         A     #LOG_1;
         JU    Fehe;
   //
   wt1:  L     #OffsetEin;
         SLW   3;
         LAR1;
   // Datenträger vorhanden
         A     DIX[AR1, P#0.0];  //DIX42.0 Codetag present
         FP    #FP_CTPR;
         =     #IMP_CTPR;
         AN    #IMP_CTPR;  // Wenn keine pos. Flanke CT_Present, dann Sprung
         JC    wt2;
         A     #LOG_1;
         =     #DataCarrierPresent;
         JU    wt3;
   wt2:  L     #OffsetEin;
         SLW   3;
         LAR1;
         AN    DIX[AR1, P#0.0];  //DIX42.0 Wenn Kein CT_Present vom BIS
         R     #DataCarrierPresent;
   wt3:  NOP   0;
END_REGION

REGION Network 4: Auswerteeinheit rücksetzten
         O     #Reset;  // FB-Eingang Reset
         FP    #FP_Reset;  // Hilfsmerker positive Flanke
         =     #IMP_Reset;  // Impulsmerker, ist einen Zyklus "1"
         A     #IMP_Reset;
         S     #ResetAktiv;
         AN    #ResetAktiv;
         JC    M014;
         R     #LesenAktiv;
         R     #SchreibenAktiv;
         R     #SchreibKonst;
         R     #Toggle;
         R     #Error;
         L     0;
         T     #ZeigerByte;
         T     #Gesamtbyte;
         T     #ErrorCode;
         L     #OffsetEin;
         SLW   3;
         TAR1;
         AN    DIX[AR1, P#0.7];  //DIX42.7 Betriebsbereit BIS
         JC    M013;
         L     #OffsetAus;  // Offset Ausgangsarrey
         SLW   3;
         LAR1;
         L     0;
         T     DIB[AR1, P#0.0];  //DIB170 Bitleiste rücksetzen
         S     DIX[AR1, P#0.2];  //DIX170.2 Resetbit setzen
         JU    M012;
   M013: L     #OffsetAus;
         SLW   3;
         LAR1;
         L     0;
         T     DIB[AR1, P#0.0];  //DIB170 Bitleiste rücksetzen
         R     #ResetAktiv;  // Rücksetzen beendet
   M012: L     DIB[AR1, P#0.0];  //DIB170
         T     #temp;
         L     #OffsetAus;  //1. Bitleiste an Ausgangsbyte übergeben
         SLW   3;
         LAR1;
         L     #temp;
         T     DBB[AR1, P#0.0];
         L     #OffsetAus;  // Adresse 2. Bitleiste
         L     #EA_Laenge;
         +I;
         L     1;
         -I;
         SLW   3;
         LAR1;
         L     #temp;
         T     DBB[AR1, P#0.0];
         JU    m100;
   M014: NOP   0;
END_REGION

REGION Network 5: Startauslösung?
         OPN   DB[ #InstanzDB];
         L     #OffsetEin;
         SLW   3;
         LAR1;
         AN    DIX[AR1, P#0.6];  //DIX42.6 Head Fehler
         JC    star;
         O     #ResetAktiv;
         O     #Reset;
         JC    M020;
         L     #CounterHF;  // Zähler um Kabelbruch nicht sofort
         +     1;  // wirksam werden zu lassen.
         T     #CounterHF;
         L     30;
         <>I;
         JC    M020;
         L     #CounterHF;  // Zähler um Kabelbruch nicht sofort
         +     -1;  // wirksam werden zu lassen.
         T     #CounterHF;
         L     9;
         JU    Fehl;
   star: L     0;
         T     #CounterHF;
         AN    #SchreibenAktiv;
         AN    #LesenAktiv;
         AN    #ResetAktiv;
         AN    #SchreibKonst;
         AN    DIX[AR1, P#0.1];  //DIX42.1 Auftrag erkannt und begonnen
         AN    DIX[AR1, P#0.3];  //DIX42.3 Auftrag fehlerhaft/ abgebrochen
         A     DIX[AR1, P#0.7];  //DIX42.7 BIS betriebsbereit
         =     #Ready;
         A     #Start;  // FB-Eingang Start
         FP    #FP_Start;  // Hilfsmerker positive Flanke
         =     #IMP_Start;  // Impulsmerker, ist einen Zyklus "1"

         A(;
         O     #IMP_Start;  // Überwachungszeit starten
         O     DIX[AR1, P#0.1];  //DIX42.1 Auftrag angenommen
         );
         AN    DIX[AR1, P#0.3];  //DIX42.3
         AN    #Dynamic;
         L     #Watchdog;
         SD    #WD_Timer;
         AN    #WD_Timer;
         JC    M020;
         L     48;  // Überwachungszeit abgelaufen
         JU    Fehl;
   M020: AN    #LesenAktiv;
         AN    #SchreibenAktiv;
         AN    #SchreibKonst;
         A(;
         AN    #IMP_Start;
         ON    #Ready;
         O     DIX[AR1, P#0.1];  //DIX42.1
         );
         BEC;
END_REGION

REGION Network 6: Initialisieren
         O     #LesenAktiv;
         JC    Lese;
         O     #SchreibenAktiv;
         JC    Schr;
         R     #Error;
         OPN   DB[ #InstanzDB];
         L     #OffsetAus;
         SLW   3;
         LAR1;
         L     0;
         T     #ErrorCode;
         T     DIB[AR1, P#0.0];  //DIB170 1. Bitleiste rücksetzen
         A     #LOG_1;
         S     DIX[AR1, P#0.0];  //DIX170.0 Auftrag vorhanden setzten
   // Leseauftrag?
         L     #Command;  // Auftragsnummer laden
         L     1;
         <>I;
         JC    M025;
         S     #LesenAktiv;  // gleich "1" -> Leseauftrag
         L     1;
         T     DIB[AR1, P#1.0];  //DIB171
         L     #Offset_DBReceive;
         T     #ZeigerByte;
         JU    M035;
   // Schreibauftrag?
   M025: L     #Command;  // Auftragsnummer laden
         L     2;
         <>I;
         JC    M026;
         L     2;
         JU    M028;
   M026: L     #Command;
         L     18;  // gleich "12hex" -> CRC Init
         <>I;
         JC    M027;
         L     18;
         JU    M028;

   M027: L     #Command;
         L     50;  // gleich "32hex" -> Konstante Daten
         <>I;
         JC    M030;
         A     #LOG_1;
         S     #SchreibKonst;
         L     50;

   M028: A     #LOG_1;
         S     #SchreibenAktiv;  // gleich "2" -> Schreibauftrag
         T     DIB[AR1, P#1.0];  //DIB171
         L     #Offset_DBSend;
         T     #ZeigerByte;
         JU    M035;

   M030: L     49;  // ungültiger Auftrag
         JU    Fehl;

   // Erster Zyklus
   M035: AN    #ErsterZyklus;
         S     #ErsterZyklus;
         R     #Ready;
   // Berechnungen
         L     #EA_Laenge;
         L     2;  // 2 Bitleisten
         -I;
         T     #ByteProSeite;  // Nutzdaten pro Seite

         A     #SchreibKonst;
         JC    M036;

         L     #NumberOfByte;
         T     #Gesamtbyte;
         JU    M037;

   M036: L     0;
         T     #Gesamtbyte;
         L     #DB_Send;
         T     #DB_Send1;
         OPN   DB[ #DB_Send1];
         L     #ZeigerByte;
         SLW   3;
         LAR1;
         L     DBB[AR1, P#0.0];  // 1. Byte Schreibdaten
         T     #temp;
         OPN   DB[ #InstanzDB];
         L     #OffsetAus;
         SLW   3;
         LAR1;
         L     #temp;
         T     DBB[AR1, P#6.0];  // Übertrag in Ausgangspuffer
   M037: NOP   1;
END_REGION

REGION Network 7: Auftrag senden
   // Die erste Bitleiste wird gespiegelt. Auftrag (Lesen, Schreiben) wird 
   // gesendet.
   // Befehlsanhang generieren
         OPN   DB[ #InstanzDB];
         L     #StartAddress;  // Anfang des Datenträgers laden
         CAW;  // Low- und Highbyte tauschen
         T     DIW[AR1, P#2.0];  //DIW172 ins 2. und 3. Byte des Ausgangspuffers schreiben
         L     #NumberOfByte;  // Laenge des Datenträgers laden
         CAW;  // Low- und Highbyte tauschen
         T     DIW[AR1, P#4.0];  //DIW174 ins 4. und 5. Byte des Ausgangspuffers schreiben

   // Erste Bitleiste spiegeln auf letztes Byte
         L     #OffsetAus;
         SLW   3;
         LAR1;
         L     DIB[AR1, P#0.0];  // Bitleiste 1
         T     #temp;
         L     #OffsetAus;
         L     #EA_Laenge;  // Adresse 2. Bitleiste
         +I;
         L     1;
         -I;
         SLW   3;
         LAR1;
         L     #temp;  // 1.Bitleiste kopieren auf 2. Bitleiste
         T     DIB[AR1, P#0.0];
   //    Auftrag schreiben
         JU    m100;
END_REGION

REGION Network 8: Lesen
   Lese: OPN   DB[ #InstanzDB];
         L     #OffsetEin;
         SLW   3;
         LAR1;
         ON    DIX[AR1, P#0.2];  //DIX42.2 Auftrag beendet
         O     DIX[AR1, P#0.3];  //DIX42.3
         BEC;
         AN    #ErsterZyklus;
         A(;
         A     #Toggle;  // Toggle-Zustand letzter Zyklus
         A     DIX[AR1, P#0.5];  //DIX42.5 Aktuelles Toggle-Bit
         O;
         AN    #Toggle;  // Toggle-Zustand letzter Zyklus
         AN    DIX[AR1, P#0.5];  //DIX42.5 Aktuelles Toggle-Bit
         );
         JC    M075;

         L     #ByteProSeite;
         L     #Gesamtbyte;
         <=I;
         JC    M050;
         T     #LaengeByte;  // Nutzdaten kleiner Nutzdaten pro Seite
         JU    M055;
   M050: L     #ByteProSeite;
         T     #LaengeByte;  // Nutzdaten größer gleich Nutzdaten pro Seite
   M055: L     #DB_Receive;
         T     #DB_Empf1;
         L     0;
         T     #schleife;  // Schleifenzähler rücksetzen
   lp3:  L     #schleife;
         L     #OffsetEin;
         +I;
         L     1;
         +I;
         SLW   3;
         LAR1;  // Leseadresse Eingang im Pointerformat
         OPN   DB[ #InstanzDB];
         L     DBB[AR1, P#0.0];
         T     #temp;
         OPN   DB[ #DB_Empf1];
         L     #ZeigerByte;
         L     #schleife;
         +I;
         SLW   3;
         LAR1;  // Zieladresse Empfangs-DB im Pointerformat
         L     #temp;
         T     DBB[AR1, P#0.0];
         L     #schleife;
         L     1;
         +I;
         T     #schleife;
         L     #LaengeByte;
         <I;
         JC    lp3;
         JU    M070;
   M075: L     #Gesamtbyte;
         L     0;
         ==D;
         JC    m090;
         BEU;
END_REGION

REGION Network 9: Schreiben
   Schr: OPN   DB[ #InstanzDB];
         A     DIX[AR1, P#0.2];  //DIX42.2 Auftrag beendet
         JC    M080;
         ON    DIX[AR1, P#0.1];  //DIX42.1 Auftrag begonnen
         O     DIX[AR1, P#0.3];  //DIX42.3 Auftrag Fehler
         BEC;
         A(;
         A     #Toggle;  // Toggle-Zustand letzter Zyklus
         A     DIX[AR1, P#0.5];  //DIX42.5 Aktuelles Toggle-Bit
         O;
         AN    #Toggle;  // Toggle-Zustand letzter Zyklus
         AN    DIX[AR1, P#0.5];  //DIX42.5 Aktuelles Toggle-Bit
         );
         BEC;

         L     #ByteProSeite;
         L     #Gesamtbyte;
         <=I;
         JC    M150;
         T     #LaengeByte;  // Nutzdaten kleiner Nutzdaten pro Seite
         JU    M155;
   M150: L     #ByteProSeite;
         T     #LaengeByte;  // Nutzdaten größer gleich Nutzdaten pro Seite
   //Nutzdaten in Ziel-DB uebertragen
   M155: L     #DB_Send;
         T     #DB_Send1;
         OPN   DB[ #DB_Send1];
         L     0;
         T     #schleife;
   lp5:  L     #ZeigerByte;
         L     #schleife;
         +I;
         SLW   3;
         LAR1;
         OPN   DB[ #DB_Send1];
         L     DBB[AR1, P#0.0];
         T     #temp;
         L     #OffsetAus;
         L     1;
         +I;
         L     #schleife;
         +I;
         SLW   3;
         LAR1;
         L     #temp;
         OPN   DB[ #InstanzDB];
         T     DBB[AR1, P#0.0];
         L     #schleife;
         L     1;
         +I;
         T     #schleife;
         L     #LaengeByte;
         <I;
         JC    lp5;
         JU    M070;
END_REGION

REGION Network 10: schreiben/ lesen
   M070: L     #OffsetEin;
         SLW   3;
         LAR1;
         L     #Gesamtbyte;  //Bytes die noch uebertragen werden müssen
         L     #LaengeByte;  //Bytes die in diesem Zyklus uebertragen wurden
         -I;  //Bytes hinzuaddieren
         T     #Gesamtbyte;

         L     #ZeigerByte;  // Zielbyte erhöhen um Nutzdatenlaenge des E/A-Bereichs
         L     #LaengeByte;
         +I;
         T     #ZeigerByte;

         OPN   DB[ #InstanzDB];
         A     DIX[AR1, P#0.5];  //DIX42.5
         =     #Toggle;  // Toggle-Zustand speichern
         L     #OffsetAus;
         SLW   3;
         LAR1;
         AN    DIX[AR1, P#0.6];
         =     DIX[AR1, P#0.6];  // Toggle-Bit invertieren im Instanz-DB 1. Bitleiste
         L     DIB[AR1, P#0.0];
         T     DIB[AR1, P#31.0];  // Bitleiste 1 kopieren in Bitleiste 2

         A     #ErsterZyklus;
         R     #ErsterZyklus;
         JU    m100;  // Übertragung noch nicht beendet
   M080: L     #OffsetEin;
         SLW   3;
         LAR1;
         AN    DIX[AR1, P#0.2];  // Auftrag Ende
         BEC;
   m090: L     #OffsetAus;
         SLW   3;
         LAR1;
         A     #LOG_1;
         R     #LesenAktiv;
         R     #SchreibenAktiv;
         R     #SchreibKonst;
         R     #Toggle;
         R     DIX[AR1, P#0.0];  // Auftrag vorhanden rücksetzten

         L     #OffsetAus;  // Auftrag vorhanden rücksetzen 1. Bitleiste
         SLW   3;
         LAR1;
         L     0;
         T     DBB[AR1, P#0.0];

         L     #OffsetAus;  // Auftrag vorhanden rücksetzen 2. Bitleiste
         L     #EA_Laenge;
         +I;
         L     1;
         -I;
         SLW   3;
         LAR1;
         L     0;
         T     DBB[AR1, P#0.0];
         JU    m100;
END_REGION

REGION Network 11: Fehler eintragen
   Fehl: T     #ErrorCode;
   Fehe: L     #Offset;
         SLW   3;
         LAR1;
         S     #Error;
         R     #Ready;
         A     #FP_Start;
         =     #Sp_start;
         L     0;
         T     DBD[AR1, P#30.0];  //DBD30
         T     DBD[AR1, P#34.0];  //DIB34
         T     DBD[AR1, P#38.0];  //DIB38
         A     #Sp_start;
         =     #FP_Start;
         JU    m090;
END_REGION

REGION Network 12: Ausgangsdaten übertragen
   m100: CALL  DPWR_DAT
         ( LADDR   := #IOAddress,
           RECORD  := #SeiteAusgang,
           RET_VAL := #ret
         );
         BEU;
END_REGION
END_FUNCTION_BLOCK

// folder: 06_Errors/01_Function

FUNCTION_BLOCK "FB600_Status.MotorDePasso"   // FB600, SCL
{ S7_Optimized_Access := 'FALSE' }
VERSION : 0.1
   VAR_INPUT
      In_DriveEnabled : Bool;   // Sinal do drive habilitado
      In_Ready : Bool;   // Sinal de estado OK do motor de passo
      In_Warning : Bool;   // Sinal de estado atenção do motor de passo
      In_Fault : Bool;   // Sinal de estado falha do motor de passo
      In_SupplyVoltPresent : Bool;   // Sinal de tensão presente
      In_DragError : Bool;   // Sinal de erro execução de movimento
      In_HomingValid : Bool;   // Sinal de homming valido
      In_StrokeLimitReached : Bool;   // Sinal de limite de giro atingido
      In_ActualPosition : DInt;   // Valor da posição atual
   END_VAR
   VAR_OUTPUT
      Out_Mensagens : String;   // Mensagens
      Out_NumeroErro : Byte;   // Numero do Erro/Sinal/Falha
   END_VAR
   VAR
      S_NumeroErro : Int;
   END_VAR
BEGIN

   (*
   BLOCO QUE CONTROLA AS MENSAGENS MOSTRADA AO OPERADOR NA IHM
   *) 

   IF #In_Warning THEN
       #Out_Mensagens := 'MOTOR EM MODO DE ATENÇÃO';
       #S_NumeroErro := 2;
   ELSIF #In_Fault THEN
       #Out_Mensagens := 'FALHA NO MOTOR';
       #S_NumeroErro := 3;
   ELSIF NOT #In_DriveEnabled AND NOT #In_Ready AND NOT #In_Warning AND NOT #In_Fault AND NOT #In_SupplyVoltPresent THEN
       #Out_Mensagens := 'MOTOR DE PASSO FORA DA REDE';
       #S_NumeroErro := 4;
   ELSIF NOT #In_DriveEnabled AND NOT #In_Ready AND NOT #In_Warning AND NOT #In_Fault AND #In_SupplyVoltPresent THEN
       #Out_Mensagens := 'MOTOR DE PASSO NÃO RECEBE COMANDOS';
       #S_NumeroErro := 8;
   ELSIF NOT #In_HomingValid THEN
       #Out_Mensagens := 'NECESSARIO REALIZAR O HOMING DO MOTOR';
       #S_NumeroErro := 5;
   ELSIF #In_DragError THEN
       #Out_Mensagens := 'ERRO NA MOVIMENTAÇÃO';
       #S_NumeroErro := 6;
   ELSIF #In_StrokeLimitReached THEN
       #Out_Mensagens := 'LIMITE DE GIRO ALCANÇADO';
       #S_NumeroErro := 7;
   ELSIF #In_DriveEnabled AND #In_Ready AND NOT #In_Warning AND NOT #In_Fault AND #In_SupplyVoltPresent THEN
       #Out_Mensagens := 'MOTOR DE PASSO DA FESTO OK';
       #S_NumeroErro := 1;
   END_IF;

   #Out_NumeroErro := INT_TO_BYTE(#S_NumeroErro);
END_FUNCTION_BLOCK

FUNCTION_BLOCK "FB601_Status.PGV"   // FB601, SCL
{ S7_Optimized_Access := 'FALSE' }
VERSION : 0.1
   VAR_INPUT
      In_ERR : Bool;   // Error Message, See Error Codes
      In_NP : Bool;   // No Absolute Position
      In_WRN : Bool;   // Warning Present, See Warning Module
      In_CA : Bool;   // Control Code Detected
      In_FR : Bool;   // Reserved
      In_FL : Bool;   // Follow Right-hand lane
      In_NL : Bool;   // Follow Left-hand lane
      In_RP : Bool;   // No lane detected
      In_TA : Bool;   // Relative Position
      In_PositionData_Y : Int;   // Valor da posição Y
      In_PositionData_X : Int;   // Valor da posição X
      In_PositionData_Z : Int;   // Valor da posição Z
      In_AngleData : Int;   // Angulo
      "In_DataMatrix.CCStatus" : Byte;   // Bit field LSB, Number of detected lanes
      "In_DataMatrix.CCNumber" : Word;   // Bit field MSB, Number of detected lanes
      "In_DataMatrix.TagNumber" : DWord;   // Data Matrix tag present
      In_BitmaskWarning : Word;   // Sinal de Warning
      In_ErrorNumber : Word;   // Numero de erro
      "In_Warning.Monitoring" : Word;   // Sinal de Warning
      "In_Error.Monitoring" : Word;   // Numero de erro
   END_VAR
   VAR_OUTPUT
      Out_Mensagens : String;   // Mensagens
      Out_NumeroErro : Byte;   // Numero do Erro/Sinal/Falha
   END_VAR
   VAR
      S_Mensagens : String;   // Memoria de mensagens
      S_Warnings : Int;   // Memoria de sinal de warning
      S_Errors : Int;   // Memoria de sinal de Erro
      S_Warning_Byte : Int;   // Memoria de sinal de warning
      S_NumeroErro : Int;   // Memoria de sinal de Erro
   END_VAR
BEGIN
   (*
   BLOCO QUE CONTROLA AS MENSAGENS MOSTRADA AO OPERADOR NA IHM
   *) 

   //Converte Word para int 
   #S_Warnings := WORD_TO_INT(#In_BitmaskWarning);
   #S_Errors := WORD_TO_INT(#In_ErrorNumber);
   #S_Warning_Byte := WORD_TO_BYTE(#In_BitmaskWarning);

   //Verifica se não existe algum erro e verifica se não existe algum alerta, então:
   IF NOT #In_ERR AND NOT #In_WRN THEN
       IF NOT #In_TA AND #In_PositionData_Y = 0
           AND #In_AngleData = 0 THEN
           #S_Mensagens := 'PGV FORA DA REDE';
           #S_NumeroErro := 2;
           ;
       ELSIF NOT #In_NP AND #In_PositionData_Y = 999
           AND #In_AngleData = 999 THEN
           #S_Mensagens := 'AGV FORA DA ROTA';
           #S_NumeroErro := 3;
       ELSIF #In_CA THEN
           #S_Mensagens := 'CODIGO DE CONTROLE DETECTADO';
           #S_NumeroErro := 4;
           ;
       ELSIF #In_FR THEN
           #S_Mensagens := 'SIGA A LINHA A DIREITA';
           #S_NumeroErro := 5;
           ;
       ELSIF #In_FL THEN
           #S_Mensagens := 'SIGA A LINHA A ESQUERDA';
           #S_NumeroErro := 6;
           ;
       ELSIF #In_NL THEN
           #S_Mensagens := 'A LINHA NÃO FOI DETECTADA';
           #S_NumeroErro := 7;
           ;
       ELSIF #In_RP THEN
           #S_Mensagens := 'POSICIONAMENTO RELATIVO';
           #S_NumeroErro := 8;
           ;

       ELSE
           #S_Mensagens := 'PGV OK';
           #S_NumeroErro := 1;
       END_IF;
       ;



   ELSIF #In_WRN THEN
       CASE #S_Warnings OF
           0:
               #S_Mensagens := 'UM CODIGO NON-PGV(QR CODE) FOI ENCONTRADO';
           1:
               #S_Mensagens := 'FITA NÃO ENCONTRADA';
           2:
               #S_Mensagens := 'PGV PERTO DA FITA';
           4:
               #S_Mensagens := 'PGV LONGE DA FITA';
           8:
               #S_Mensagens := 'FITA MUITO LARGA';
           16:
               #S_Mensagens := 'FITA MUITO FINA';
           32:
               #S_Mensagens := 'PGV DESALINHADO EM RELAÇÃO A FITA';
           64:
               #S_Mensagens := 'POUCO CONTRASTE NA FITA';
           128:
               #S_Mensagens := 'NECESSARIOA REPARAR A FITA';
           255:
               #S_Mensagens := 'TEMPERATURA MUITO ALTA';

       END_CASE;

       ;


   ELSIF #In_ERR THEN
       CASE #S_Errors OF
           2:
               #S_Mensagens := 'Impossivel determinar um posicao limpa'; //Diferença entre QR Code é muito grande ou Distancia de codigo esta incorreta
               ;
           5:
               #S_Mensagens := 'SEM DECISÃO DE DIREÇÃO HABILITADA';
           1000:
               #S_Mensagens := 'ERRO INTERNO';
               ;
       END_CASE;
       ;
   ELSE
       #S_Mensagens := 'PGV OK';
   END_IF;


   #Out_Mensagens BLKMOV #S_Mensagens;
   #Out_NumeroErro := INT_TO_BYTE(#S_NumeroErro);
END_FUNCTION_BLOCK

FUNCTION_BLOCK "FB602_Status.Rfid"   // FB602, SCL
{ S7_Optimized_Access := 'FALSE' }
VERSION : 0.1
   VAR_INPUT
      In_Posto : Int;   // Valor do Posto que o AGV esta
      In_Comando : Int;   // Valor do Comando
      In_Velocidade : Int;   // Valor da Velocidade
      In_Linha : Int;   // Valor da linha
      In_Tag_Presente : Bool;   // Sinal de Tag presente
      In_Error : Bool;   // Sinal de Erro
      In_Code_Error : Int;   // Codigo de Error
      In_Ready : Bool;   // Sinal de tudo OK
   END_VAR
   VAR_OUTPUT
      Out_Mensagem : String;   // Mensagens
      Out_ErroNumero : Byte;   // Numero do Erro/Sinal/Falha
   END_VAR
   VAR
      ErrorCodeString : String;
   END_VAR
BEGIN
   (*
   BLOCO QUE CONTROLA AS MENSAGENS MOSTRADA AO OPERADOR NA IHM
   *) 

   //Realiza a tranformação da informação de int para string
   #ErrorCodeString := INT_TO_STRING("DB600_AgvSinais".RFID.Code_Error);


   IF "DB1_DatabaseAgv".RFID.Error OR "DB1_DatabaseAgv".RFID.Fault OR ("DB1_DatabaseAgv".RFID.CodigoErro <> 0) THEN
       #Out_Mensagem := CONCAT(IN1 := 'FALHA NO RFID, O COD DO ERRO É ', IN2 := #ErrorCodeString);
       #Out_ErroNumero:= 2;
   ELSIF "IOLink_StatusAGV" = 16#0000 THEN
       #Out_Mensagem  := 'RFID FORA DA REDE';
       #Out_ErroNumero := 3;
   ELSIF "DB600_AgvSinais".RFID.Ready AND NOT #In_Tag_Presente  THEN
       #Out_Mensagem := 'RFID OK';
       #Out_ErroNumero := 1;
   ELSIF "DB600_AgvSinais".RFID.Tag_Presente THEN
       #Out_Mensagem := 'CARTÃO RFID DETECTADO';
       #Out_ErroNumero := 4;
   ELSIF NOT "DB600_AgvSinais".RFID.Ready THEN
       #Out_Mensagem := 'A ANTENA RFID NÃO ESTA PRONTO PARA LER TAGS';
       #Out_ErroNumero := 5;
   ELSE
       #Out_Mensagem := 'RFID NOT OK!';
       #Out_ErroNumero := 6;
   END_IF;
END_FUNCTION_BLOCK

FUNCTION_BLOCK "FB603_StatusGeralAgv"   // FB603, SCL
TITLE = FB603_StatusGeralAgv
{ S7_Optimized_Access := 'FALSE' }
AUTHOR : ssbjvq
FAMILY : AGV_KD
VERSION : 0.1
// Bloco responsavel por gerenciar todos os erros do AGV
   VAR
      FB60_StatusSteppingMotor_Instance : "FB600_Status.MotorDePasso";
      FB61_StatusPGV_Instance : "FB601_Status.PGV";
      FB62_StatusRfid_Instance : "FB602_Status.Rfid";
      ERRO : Int;   // Valor de erro do bloco de aquisição da hora atual
      S_NumeroErro : Int;   // Memoria de valor do Erro que irá para IHM
   END_VAR
BEGIN
   (*
   BLOCO QUE CONTROLA AS MENSAGENS MOSTRADA AO OPERADOR NA IHM
   *) 

   REGION BlocoDeErrosMotor
       #FB60_StatusSteppingMotor_Instance(In_DriveEnabled := "DB600_AgvSinais".Stepping_Motor.Outputs.DriveEnabled,
                                          In_Ready := "DB600_AgvSinais".Stepping_Motor.Outputs.Ready,
                                          In_Warning := "DB600_AgvSinais".Stepping_Motor.Outputs.Warning,
                                          In_Fault := "DB600_AgvSinais".Stepping_Motor.Outputs.Fault,
                                          In_SupplyVoltPresent := "DB600_AgvSinais".Stepping_Motor.Outputs.SupplyVoltPresent,
                                          In_DragError := "DB600_AgvSinais".Stepping_Motor.Outputs.DragError,
                                          In_HomingValid := "DB600_AgvSinais".Stepping_Motor.Outputs.HomingValid,
                                          In_StrokeLimitReached := "DB600_AgvSinais".Stepping_Motor.Outputs.StrokeLimitReached,
                                          In_ActualPosition := "DB600_AgvSinais".Stepping_Motor.Outputs.ActualPosition,
                                          Out_Mensagens => "DB600_AgvSinais".Stepping_Motor.Mensagem,
                                          Out_NumeroErro => "DB700_EnviaDados".Dados."Erros.MotorPasso");
   END_REGION

   REGION BlocoDeLeituraDoPgv
       #FB61_StatusPGV_Instance(In_ERR := "DB600_AgvSinais".PGV.ERR,
                                In_NP := "DB600_AgvSinais".PGV.NP,
                                In_WRN := "DB600_AgvSinais".PGV.WRN,
                                In_CA := "DB600_AgvSinais".PGV.CA,
                                In_FR := "DB600_AgvSinais".PGV.FR,
                                In_FL := "DB600_AgvSinais".PGV.FL,
                                In_NL := "DB600_AgvSinais".PGV.NL,
                                In_RP := "DB600_AgvSinais".PGV.RP,
                                In_TA := "DB600_AgvSinais".PGV.TA,
                                In_PositionData_Y := "DB600_AgvSinais".PGV.PositionData_Y,
                                In_PositionData_X := "DB600_AgvSinais".PGV.PositionData_X,
                                In_PositionData_Z := "DB600_AgvSinais".PGV.PositionData_Z,
                                In_AngleData := "DB600_AgvSinais".PGV.AngleData,
                                "In_DataMatrix.CCStatus" := "DB600_AgvSinais".PGV."DataMatrix.CCStatus",
                                "In_DataMatrix.CCNumber" := "DB600_AgvSinais".PGV."DataMatrix.CCNumber",
                                "In_DataMatrix.TagNumber" := "DB600_AgvSinais".PGV."DataMatrix.TagNumber",
                                In_BitmaskWarning := "DB600_AgvSinais".PGV.BitmaskWarning,
                                In_ErrorNumber := "DB600_AgvSinais".PGV.ErrorNumber,
                                "In_Warning.Monitoring" := "DB600_AgvSinais".PGV."OUT_Warning.Monitoring",
                                "In_Error.Monitoring" := "DB600_AgvSinais".PGV."OUT_Error.Monitoring",
                                Out_Mensagens => "DB600_AgvSinais".PGV.Mensagem,
                                Out_NumeroErro => "DB700_EnviaDados".Dados."Erros.Pgv");

                             END_REGION

   REGION BlocoDeErrosdoRFID
       #FB62_StatusRfid_Instance(In_Posto := "DB600_AgvSinais".RFID.Posto,
                                 In_Comando := "DB600_AgvSinais".RFID.Comando,
                                 In_Velocidade := "DB600_AgvSinais".RFID.Velocidade,
                                 In_Linha := "DB600_AgvSinais".RFID.Linha,
                                 In_Tag_Presente := "DB600_AgvSinais".RFID.Tag_Presente,
                                 In_Error := "DB600_AgvSinais".RFID.Error,
                                 In_Code_Error := "DB600_AgvSinais".RFID.Code_Error,
                                 In_Ready := "DB600_AgvSinais".RFID.Ready,
                                 Out_Mensagem => "DB600_AgvSinais".RFID.Mensagem,
                                 Out_ErroNumero => "DB700_EnviaDados".Dados."Erros.Rfid");

   END_REGION

   REGION MovimentaçãoDeDados
       // Esta parte realiza a movimentação dos dados para a DB que a IHM consulta para ver os estados

       REGION Cartões de Entrada
           //Cartões de Entrada
           "DB600_AgvSinais".Inputs."8DI_24V"."I0.0" := "DI_BotaoStart";
           "DB600_AgvSinais".Inputs."8DI_24V"."I0.1" := "DI_Emergencia";
           "DB600_AgvSinais".Inputs."8DI_24V"."I0.2" := "DI_Resevado";
           "DB600_AgvSinais".Inputs."8DI_24V"."I0.3" := "DI_Resevado_1";
           "DB600_AgvSinais".Inputs."8DI_24V"."I0.4" := "DI_ScannerWarning";
           "DB600_AgvSinais".Inputs."8DI_24V"."I0.5" := "DI_ScannerSafety";
           "DB600_AgvSinais".Inputs."8DI_24V"."I0.6" := "DI_Resevado_2";
           "DB600_AgvSinais".Inputs."8DI_24V"."I0.7" := "DI_Resevado_3";
       END_REGION
       REGION Cartões de Saida
           //Digital
           "DB600_AgvSinais".Outputs."8DO_24V"."Q0.0" := "DO_Reservado";
           "DB600_AgvSinais".Outputs."8DO_24V"."Q0.1" := "DO_Reservado_1";
           "DB600_AgvSinais".Outputs."8DO_24V"."Q0.2" := "DO_Motor.Frente";
           "DB600_AgvSinais".Outputs."8DO_24V"."Q0.3" := "DO_Motor.Tras";
           "DB600_AgvSinais".Outputs."8DO_24V"."Q0.4" := "DO_Scanner.Zone1";
           "DB600_AgvSinais".Outputs."8DO_24V"."Q0.5" := "DO_Giroflex";
           "DB600_AgvSinais".Outputs."8DO_24V"."Q0.6" := "DO_Scanner.Zone2";
           "DB600_AgvSinais".Outputs."8DO_24V"."Q0.7" := "DO_LuzReset";
           //Analogico
           "DB600_AgvSinais".Outputs."2AO x U ST".QW750 := "AO_MotorTracao";
           "DB600_AgvSinais".Outputs."2AO x U ST".QW752 := "AO_Reservado";
       END_REGION
       REGION RFID
           //RFID
           "DB600_AgvSinais".RFID.Posto := "DB1_DatabaseAgv".RFID.Posto;
           "DB600_AgvSinais".RFID.Comando := "DB1_DatabaseAgv".RFID.Comando;
           "DB600_AgvSinais".RFID.Velocidade := "DB1_DatabaseAgv".RFID.Velocidade;
           "DB600_AgvSinais".RFID.Linha := "DB1_DatabaseAgv".RFID.Processo;
           "DB600_AgvSinais".RFID.Tag_Presente := "DB1_DatabaseAgv".RFID.TagPresente;
           "DB600_AgvSinais".RFID.Error := "DB1_DatabaseAgv".RFID.Error;
           "DB600_AgvSinais".RFID.Code_Error := "DB1_DatabaseAgv".RFID.CodigoErro;
           "DB600_AgvSinais".RFID.Ready := "DB1_DatabaseAgv".RFID.Ready;
           "DB1_DatabaseAgv".RFID.Posto := "DB3_Memorias".Rfid.Posto;
           "DB1_DatabaseAgv".RFID.Comando := "DB3_Memorias".Rfid.Comando;
           "DB1_DatabaseAgv".RFID.Processo := "DB3_Memorias".Rfid.Linha;
           "DB500_SinaisIhm".VelocidadeAtual := ("DB1_DatabaseAgv".Saidas.VelocidadeMotorTracao / 1000);

       END_REGION
       REGION Stepping Motor
           //Stepping Motor
           //Input
           "DB600_AgvSinais".Stepping_Motor.Inputs.Enabla_Drive := "DB1_DatabaseAgv".MotorDePasso.Inputs.EnableDrive;
           "DB600_AgvSinais".Stepping_Motor.Inputs.Stop := "DB1_DatabaseAgv".MotorDePasso.Inputs.Stop;
           "DB600_AgvSinais".Stepping_Motor.Inputs."Start Task" := "DB1_DatabaseAgv".MotorDePasso.Inputs.StartTask;
           "DB600_AgvSinais".Stepping_Motor.Inputs.Opm := "DB1_DatabaseAgv".MotorDePasso.Inputs.OPM;
           "DB600_AgvSinais".Stepping_Motor.Inputs.Brake := "DB1_DatabaseAgv".MotorDePasso.Inputs.Brake;
           //Output
           "DB600_AgvSinais".Stepping_Motor.Outputs.DriveEnabled := "DB1_DatabaseAgv".MotorDePasso.OutPuts.DriveEnabled;
           "DB600_AgvSinais".Stepping_Motor.Outputs.Ready := "DB1_DatabaseAgv".MotorDePasso.OutPuts.Ready;
           "DB600_AgvSinais".Stepping_Motor.Outputs.Warning := "DB1_DatabaseAgv".MotorDePasso.OutPuts.Warning;
           "DB600_AgvSinais".Stepping_Motor.Outputs.Fault := "DB1_DatabaseAgv".MotorDePasso.OutPuts.Fault;
           "DB600_AgvSinais".Stepping_Motor.Outputs.SupplyVoltPresent := "DB1_DatabaseAgv".MotorDePasso.OutPuts.SupplyVoltPresent;
           "DB600_AgvSinais".Stepping_Motor.Outputs.DragError := "DB1_DatabaseAgv".MotorDePasso.OutPuts.DragError;
           "DB600_AgvSinais".Stepping_Motor.Outputs.HomingValid := "DB1_DatabaseAgv".MotorDePasso.OutPuts.HomingValid;
           "DB600_AgvSinais".Stepping_Motor.Outputs.StrokeLimitReached := "DB1_DatabaseAgv".MotorDePasso.OutPuts.StrokeLimitReached;
           "DB600_AgvSinais".Stepping_Motor.Outputs.ActualPosition := "DB1_DatabaseAgv".MotorDePasso.OutPuts.ActualPosition;

       END_REGION
       REGION PGV        
           //PGV
           "DB600_AgvSinais".PGV.ERR := "DB1_DatabaseAgv".PGV.Module2.Status.ERR;
           "DB600_AgvSinais".PGV.NP := "DB1_DatabaseAgv".PGV.Module2.Status.NP;
           "DB600_AgvSinais".PGV.WRN := "DB1_DatabaseAgv".PGV.Module2.Status.WRN;
           "DB600_AgvSinais".PGV.CA := "DB1_DatabaseAgv".PGV.Module2.Status.CC;
           "DB600_AgvSinais".PGV.FR := "DB1_DatabaseAgv".PGV.Module2.Status.FR;
           "DB600_AgvSinais".PGV.FL := "DB1_DatabaseAgv".PGV.Module2.Status.FL;
           "DB600_AgvSinais".PGV.NL := "DB1_DatabaseAgv".PGV.Module2.Status.NL;
           "DB600_AgvSinais".PGV.RP := "DB1_DatabaseAgv".PGV.Module2.Status.RP;
           "DB600_AgvSinais".PGV.TA := "DB1_DatabaseAgv".PGV.Module2.Status.TA;

           "DB600_AgvSinais".PGV.PositionData_Y := DWORD_TO_INT("DB1_DatabaseAgv".PGV.Module2.PositionY);
           "DB600_AgvSinais".PGV.PositionData_X := DWORD_TO_INT("DB1_DatabaseAgv".PGV.Module2.PositionX);
           "DB600_AgvSinais".PGV.PositionData_Z := DWORD_TO_INT("DB1_DatabaseAgv".PGV.Module2.PositionZ);
           "DB600_AgvSinais".PGV.AngleData := DWORD_TO_INT("DB1_DatabaseAgv".PGV.Module2.Angle);
           "DB600_AgvSinais".PGV.BitmaskWarning := "DB1_DatabaseAgv".PGV.Module5.BitmaskWarning;
           "DB600_AgvSinais".PGV.ErrorNumber := "DB1_DatabaseAgv".PGV.Module5.ErroNumber;
       END_REGION
       REGION DataHora
           //Date e Hora
           #ERRO := RD_SYS_T("DB600_AgvSinais".DateHora);

       END_REGION



   END_REGION

   REGION LogicaMensagens

       //Mensagens de falha do AGV

       // 0000 0000  0000 0000     
       IF NOT "DB600_AgvSinais".Inputs."8DI_24V"."I0.5" THEN
           "DB600_AgvSinais".Mensagens_Global := 'AREA DE SEGURANÇA DO SCANNER INFRINGIDA';
           // 0000 0001  0000 0000  
           "DB600_AgvSinais".Alarms[0] := 8;
           #S_NumeroErro := 2;

       ELSIF "DB600_AgvSinais".Inputs."8DI_24V"."I0.1" THEN
           "DB600_AgvSinais".Mensagens_Global := 'EMERGENCIA ACIONADO!!!';
           #S_NumeroErro := 9;
           // 0004 0000  0000 0000  
           "DB600_AgvSinais".Alarms[0] := 16;
       ELSIF "DB600_AgvSinais".Stepping_Motor.Outputs.Fault OR (NOT "DB600_AgvSinais".Stepping_Motor.Outputs.DriveEnabled AND "DB600_AgvSinais".Stepping_Motor.Outputs.SupplyVoltPresent) THEN
           "DB600_AgvSinais".Mensagens_Global := 'FALHA NO MOTOR DE PASSO';
           // 0001 0000  0000 0000  
           "DB600_AgvSinais".Alarms[0] := 32;
           #S_NumeroErro := 3;
       ELSIF NOT "DB600_AgvSinais".Stepping_Motor.Outputs.DriveEnabled
           AND NOT "DB600_AgvSinais".Stepping_Motor.Outputs.Ready
           AND NOT "DB600_AgvSinais".Stepping_Motor.Outputs.Warning
           AND NOT "DB600_AgvSinais".Stepping_Motor.Outputs.Fault
           AND NOT "DB600_AgvSinais".Stepping_Motor.Outputs.SupplyVoltPresent THEN
           // 0000 0000  0000 0010  
           "DB600_AgvSinais".Alarms[0] := 512;
           "DB600_AgvSinais".Mensagens_Global := 'MOTOR DE PASSO FORA DA REDE';
           #S_NumeroErro := 4;


       ELSIF "IOLink_StatusAGV" = 16#0000 THEN
           "DB600_AgvSinais".Mensagens_Global := 'RFID FORA DA REDE';
           // 0000 0000  0000 0100  
           "DB600_AgvSinais".Alarms[0] := 128;
           #S_NumeroErro := 5;

       ELSIF NOT "DB600_AgvSinais".PGV.NP
           AND "DB600_AgvSinais".PGV.PositionData_Y = 999
           AND "DB600_AgvSinais".PGV.AngleData = 999 THEN
           "DB600_AgvSinais".Mensagens_Global := 'AGV FORA DA ROTA';
           #S_NumeroErro := 6;
           // 0000 0001  0000 0000  
           "DB600_AgvSinais".Alarms[0] := 2;
       ELSIF "DB600_AgvSinais".PGV.PositionData_Y = 0
           AND "DB600_AgvSinais".PGV.AngleData = 0 THEN
           "DB600_AgvSinais".Mensagens_Global := 'PGV FORA DA REDE';
           #S_NumeroErro := 7;
           // 0000 0000  0000 0100  
           "DB600_AgvSinais".Alarms[0] := 256;
       ELSIF "DB600_AgvSinais".Inputs."8DI_24V"."I0.4" THEN
           "DB600_AgvSinais".Mensagens_Global := 'AREA DE ATENÇÃO DO SCANNER INFRINGIDA';
           #S_NumeroErro := 8;
           // 0000 0010  0000 0000  
           "DB600_AgvSinais".Alarms[0] := 4;

       ELSIF ("DB500_SinaisIhm".ConectarTakt = 0) AND "DB500_SinaisIhm".ConexaoTakt THEN
           "DB600_AgvSinais".Mensagens_Global := 'SEM COMUNICAÇÃO COM O TAKT';
           "DB600_AgvSinais".Alarms[0] := 1024;
           #S_NumeroErro := 11;
       ELSIF "DB701_RecebeDados".Dados.EmergenciaECU THEN
           "DB600_AgvSinais".Mensagens_Global := 'EMERGENCIA ACIONADO NA LINHA DE ECU';
           "DB600_AgvSinais".Alarms[0] := 2048;
           #S_NumeroErro := 12;
   (* ELSIF   THEN
       "DB600_AgvSinais".Mensagens_Global := 'CHAVE DO MOTOR DE TRAÇÂO DESLIGADA';
       "DB600_AgvSinais".Alarms[0] := 64;
        #S_NumeroErro := 10;
    *)
       ELSIF "DB1_DatabaseAgv".RFID.Error OR "DB1_DatabaseAgv".RFID.Fault OR ("DB1_DatabaseAgv".RFID.CodigoErro <> 0) OR NOT "DB600_AgvSinais".RFID.Ready THEN
           "DB600_AgvSinais".Mensagens_Global := 'FALHA NO RFID';
           "DB600_AgvSinais".Alarms[0] := 4096;
           #S_NumeroErro := 13;
       ELSE
           "DB600_AgvSinais".Mensagens_Global := 'AGV OK';
           "DB600_AgvSinais".Alarms[0] := 0;
           #S_NumeroErro := 1;

       END_IF;

       "DB700_EnviaDados".Dados."Erros.Agv" := INT_TO_BYTE(#S_NumeroErro);
   END_REGION
END_FUNCTION_BLOCK

// folder: 06_Errors/03_OB

ORGANIZATION_BLOCK "I/O_FLT1"   // OB82, LAD
TITLE = "I/O Point Fault"
{ S7_Optimized_Access := 'FALSE' }
VERSION : 0.1
   VAR_TEMP
      OB82_EV_CLASS : Byte;   // 16#39, Event class 3, Entering event state, Internal fault event
      OB82_FLT_ID : Byte;   // 16#XX, Fault identifcation code
      OB82_PRIORITY : Byte;   // Priority of OB Execution
      OB82_OB_NUMBR : Byte;   // 82 (Organization block 82, OB82)
      OB82_RESERVED_1 : Byte;   // Reserved for system
      OB82_IO_FLAG : Byte;   // Input (01010100), Output (01010101)
      OB82_MDL_ADDR : Word;   // Base address of module with fault
      OB82_MDL_DEFECT : Bool;   // Module defective
      OB82_INT_FAULT : Bool;   // Internal fault
      OB82_EXT_FAULT : Bool;   // External fault
      OB82_PNT_INFO : Bool;   // Point information
      OB82_EXT_VOLTAGE : Bool;   // External voltage low
      OB82_FLD_CONNCTR : Bool;   // Field wiring connector missing
      OB82_NO_CONFIG : Bool;   // Module has no configuration data
      OB82_CONFIG_ERR : Bool;   // Module has configuration error
      OB82_MDL_TYPE : Byte;   // Type of module
      OB82_SUB_MDL_ERR : Bool;   // Sub-Module is missing or has error
      OB82_COMM_FAULT : Bool;   // Communication fault
      OB82_MDL_STOP : Bool;   // Module is stopped
      OB82_WTCH_DOG_FLT : Bool;   // Watch dog timer stopped module
      OB82_INT_PS_FLT : Bool;   // Internal power supply fault
      OB82_PRIM_BATT_FLT : Bool;   // Primary battery is in fault
      OB82_BCKUP_BATT_FLT : Bool;   // Backup battery is in fault
      OB82_RESERVED_2 : Bool;   // Reserved for system
      OB82_RACK_FLT : Bool;   // Rack fault, only for bus interface module
      OB82_PROC_FLT : Bool;   // Processor fault
      OB82_EPROM_FLT : Bool;   // EPROM fault
      OB82_RAM_FLT : Bool;   // RAM fault
      OB82_ADU_FLT : Bool;   // ADU fault
      OB82_FUSE_FLT : Bool;   // Fuse fault
      OB82_HW_INTR_FLT : Bool;   // Hardware interupt input in fault
      OB82_RESERVED_3 : Bool;   // Reserved for system
      OB82_DATE_TIME : Date_And_Time;   // Date and time OB82 started
   END_VAR
BEGIN
END_ORGANIZATION_BLOCK

ORGANIZATION_BLOCK "I/O_FLT2"   // OB83, LAD
TITLE = "I/O Point Fault"
{ S7_Optimized_Access := 'FALSE' }
VERSION : 0.1
   VAR_TEMP
      OB83_EV_CLASS : Byte;   // 16#38/39, Event class 3, module inserted/removed (8/9)
      OB83_FLT_ID : Byte;   // 16#XX, Fault identifcation code
      OB83_PRIORITY : Byte;   // Priority of OB Execution
      OB83_OB_NUMBR : Byte;   // 83 (Organization block 83, OB83)
      OB83_RESERVED_1 : Byte;   // Reserved for system
      OB83_MDL_ID : Byte;   // Input module (01010100), Output module (01010101)
      OB83_MDL_ADDR : Word;   // Base address of module with point fault
      OB83_RACK_NUM : Int;   // Number of rack that has module with point fault
      OB83_MDL_TYPE : Word;   // Module type with point fault
      OB83_DATE_TIME : Date_And_Time;   // Date and time OB83 started
   END_VAR
BEGIN
END_ORGANIZATION_BLOCK

ORGANIZATION_BLOCK "OBNL_FLT"   // OB85, LAD
TITLE = "Organization Block (OB) Not Loaded Fault"
{ S7_Optimized_Access := 'FALSE' }
VERSION : 0.1
   VAR_TEMP
      OB85_EV_CLASS : Byte;   // 16#35 Event class 3
      OB85_FLT_ID : Byte;   // 16#XX, Fault identification code
      OB85_PRIORITY : Byte;   // Priority of OB Execution
      OB85_OB_NUMBR : Byte;   // 85 (Organization block 85, OB85)
      OB85_RESERVED_1 : Byte;   // Reserved for system
      OB85_RESERVED_2 : Byte;   // Reserved for system
      OB85_RESERVED_3 : Int;   // Reserved for system
      OB85_ERR_EV_CLASS : Byte;   // Class of event causing error
      OB85_ERR_EV_NUM : Byte;   // Number of event causing error
      OB85_OB_PRIOR : Byte;   // Priority of OB causing error
      OB85_OB_NUM : Byte;   // Number of OB causing error
      OB85_DATE_TIME : Date_And_Time;   // Date and time OB85 started
   END_VAR
BEGIN
END_ORGANIZATION_BLOCK

ORGANIZATION_BLOCK "RACK_FLT"   // OB86, LAD
TITLE = "Loss Of Rack Fault"
{ S7_Optimized_Access := 'FALSE' }
VERSION : 0.1
   VAR_TEMP
      OB86_EV_CLASS : Byte;   // 16#38/39 Event class 3
      OB86_FLT_ID : Byte;   // 16#C1/C4/C5, Fault identification code
      OB86_PRIORITY : Byte;   // Priority of OB Execution
      OB86_OB_NUMBR : Byte;   // 86 (Organization block 86, OB86)
      OB86_RESERVED_1 : Byte;   // Reserved for system
      OB86_RESERVED_2 : Byte;   // Reserved for system
      OB86_MDL_ADDR : Word;   // Base address of IM module in rack with fault
      OB86_RACKS_FLTD : Array[0..31] of Bool;   // Racks in fault
      OB86_DATE_TIME : Date_And_Time;   // Date and time OB86 started
   END_VAR
BEGIN
END_ORGANIZATION_BLOCK

ORGANIZATION_BLOCK "COMM_FLT"   // OB87, LAD
TITLE = "Communication Fault"
{ S7_Optimized_Access := 'FALSE' }
VERSION : 0.1
   VAR_TEMP
      OB87_EV_CLASS : Byte;   // 16#39 Event class 3
      OB87_FLT_ID : Byte;   // 16#XX, Fault identifcation code
      OB87_PRIORITY : Byte;   // Priority of OB Execution
      OB87_OB_NUMBR : Byte;   // 87 (Organization block 87, OB87)
      OB87_RESERVED_1 : Byte;   // Reserved for system
      OB87_RESERVED_2 : Byte;   // Reserved for system
      OB87_RESERVED_3 : Word;   // Reserved for system
      OB87_RESERVED_4 : DWord;   // Reserved for system
      OB87_DATE_TIME : Date_And_Time;   // Date and time OB87 started
   END_VAR
BEGIN
END_ORGANIZATION_BLOCK

ORGANIZATION_BLOCK "PROG_ERR"   // OB121, LAD
TITLE = "Programming Error"
{ S7_Optimized_Access := 'FALSE' }
VERSION : 0.1
   VAR_TEMP
      OB121_EV_CLASS : Byte;   // 16#25, Event class 2, Entering event state, Internal fault event
      OB121_SW_FLT : Byte;   // 16#XX Software programming fault
      OB121_PRIORITY : Byte;   // Priority of OB Execution
      OB121_OB_NUMBR : Byte;   // 121 (Organization block 121, OB121)
      OB121_BLK_TYPE : Byte;   // 16#88/8A/8B/8C/8E Type of block fault occured in
      OB121_RESERVED_1 : Byte;   // Reserved for system
      OB121_FLT_REG : Word;   // 16#XX Specific register that caused fault
      OB121_BLK_NUM : Word;   // Number of block that programming fault occured in
      OB121_PRG_ADDR : Word;   // Address in block where programming fault occured
      OB121_DATE_TIME : Date_And_Time;   // Date and time OB121 started
   END_VAR
BEGIN
END_ORGANIZATION_BLOCK

ORGANIZATION_BLOCK "MOD_ERR"   // OB122, LAD
TITLE = "Module Access Error"
{ S7_Optimized_Access := 'FALSE' }
VERSION : 0.1
   VAR_TEMP
      OB122_EV_CLASS : Byte;   // 16#29, Event class 2, Entering event state, Internal fault event
      OB122_SW_FLT : Byte;   // 16#XX Software error code
      OB122_PRIORITY : Byte;   // Priority of OB Execution
      OB122_OB_NUMBR : Byte;   // 122 (Organization block 122, OB122)
      OB122_BLK_TYPE : Byte;   // 16#88/8C/8E Type of block fault occured in
      OB122_MEM_AREA : Byte;   // Memory area where access error occured
      OB122_MEM_ADDR : Word;   // Memory address where access error occured
      OB122_BLK_NUM : Word;   // Block number in which error occured
      OB122_PRG_ADDR : Word;   // Program address where error occured
      OB122_DATE_TIME : Date_And_Time;   // Date and time OB1 started
   END_VAR
BEGIN
END_ORGANIZATION_BLOCK

// folder: 07_Takt/01_Function

FUNCTION_BLOCK "FB703_ControleTakt"   // FB703, SCL
TITLE = FB703_ControleTakt
{ S7_Optimized_Access := 'FALSE' }
AUTHOR : ssbjvq
FAMILY : AGV_KD
VERSION : 0.1
// Realiza a comunicação com o takt (Leitura e escrita)
   VAR_INPUT
      In_Dados : "EscritaTakt";
   END_VAR
   VAR_OUTPUT
      Out_Dados : "LeituraTakt";
      Out_Get_Error : Bool;
      Out_Get_Status : Word;
      Out_Set_Erro : Bool;
      Out_Set_Status : Word;
   END_VAR
   VAR
      GET_DadosTakt : GET;
      PUT_DadosTakt : PUT;
      FB704_VerificaConexãoTakt : "FB704_VerificaConexãoTakt";
   END_VAR
   // GET_DadosTakt.ID := 16#1;
BEGIN
   //------------------ Verifica Conexão com o Takt ------------------//
   #FB704_VerificaConexãoTakt("DB701_RecebeDados".Dados.WatchDog);


   //------------------ Realiza a leitura dos dados do TAKT ------------------//
   (* #GET_DadosTakt(REQ := "Clock_0.5Hz" AND "DB500_SinaisIhm".ConexaoTakt,
                  ID := 16#1,
                  ERROR => #Out_Get_Error,
                  STATUS => #Out_Get_Status,
                  ADDR_1 := P# DB200.DBX0.0 BYTE 2,
                  RD_1 := P# DB701.DBX0.0 BYTE 2); 
   *)
   (* "DB500_SinaisIhm".ConectarTakt := BOOL_TO_INT(#Out_Get_Error); *)

   //------------------ Realiza a escrita dos dados do TAKT ------------------//
   (*
   #PUT_DadosTakt(REQ:=NOT "Clock_10Hz",
                  ID:=16#1,
                  ERROR=>#Out_Set_Erro,
                  STATUS=>#Out_Set_Status,
                  ADDR_1:=P# DB10.DBX0.0 BYTE 22,
                  SD_1:=P# DB700.DBX0.0 BYTE 22);
   *)
   "DB700_EnviaDados".Dados.Emergencia := "DI_Emergencia";
   "DB700_EnviaDados".Dados.Warning := "DI_ScannerWarning";
   "DB700_EnviaDados".Dados.Safety := "DI_ScannerSafety";
   "DB700_EnviaDados".Dados.AutomaticoManual := INT_TO_BYTE("DB500_SinaisIhm".ManualAutomatico);
   "DB700_EnviaDados".Dados.VelocidadeAtual := "AO_MotorTracao";
   "DB700_EnviaDados".Dados.Posto := INT_TO_BYTE("DB1_DatabaseAgv".RFID.Posto);
   "DB700_EnviaDados".Dados.Comando := INT_TO_BYTE("DB1_DatabaseAgv".RFID.Comando);
   "DB700_EnviaDados".Dados.Velocidade := INT_TO_BYTE("DB1_DatabaseAgv".RFID.Velocidade);
   "DB700_EnviaDados".Dados.Processo := INT_TO_BYTE("DB1_DatabaseAgv".RFID.Processo);
   "DB700_EnviaDados".Dados.ConectarTakt := "DB500_SinaisIhm".ConexaoTakt;
END_FUNCTION_BLOCK

FUNCTION_BLOCK "FB704_VerificaConexãoTakt"   // FB704, SCL
TITLE = FB704_VerificaConexãoTakt
{ S7_Optimized_Access := 'FALSE' }
VERSION : 0.1
// FB704_VerificaConexãoTakt
   VAR_INPUT
      In_WatchDog : Bool;
   END_VAR
   VAR
      ClockCustomizado : "FB705_WatchdogTakt";
      TON_Conexao : TON;
   END_VAR
BEGIN

   #ClockCustomizado(In_Tempo:=T#60s);

   IF #ClockCustomizado.Out_Sinal AND #In_WatchDog THEN
       "DB701_RecebeDados".Dados.WatchDog := 0;
   END_IF;


   #TON_Conexao(IN:= NOT "DB701_RecebeDados".Dados.WatchDog,
                PT:=T#60s);

   IF  #TON_Conexao.Q THEN
       "DB500_SinaisIhm".ConectarTakt := 0;
   ELSE
       "DB500_SinaisIhm".ConectarTakt  := 1;
   END_IF;
END_FUNCTION_BLOCK

FUNCTION_BLOCK "FB705_WatchdogTakt"   // FB705, SCL
{ S7_Optimized_Access := 'FALSE' }
VERSION : 0.1
   VAR_INPUT
      In_Tempo : Time;
   END_VAR
   VAR_OUTPUT
      Out_Sinal : Bool;
      Out_NotSinal : Bool;
   END_VAR
   VAR
      TON_1 : TON;
      TON_2 : TON;
   END_VAR
BEGIN
   #TON_1(IN:=NOT #TON_2.Q,
          PT:=#In_Tempo);
   #TON_2(IN:=#TON_1.Q,
          PT:=#In_Tempo);



   #Out_Sinal := #TON_1.Q;
   #Out_NotSinal := NOT #TON_1.Q;
END_FUNCTION_BLOCK

(* ===== HMI "HMI_AGV72159" =====
system functions are stored by id; their names below are inferred from use
connection "HMI": ETHERNET, SIMATIC S7 300/400 MPI

